KUKA KRL program: MyProgram_118().src

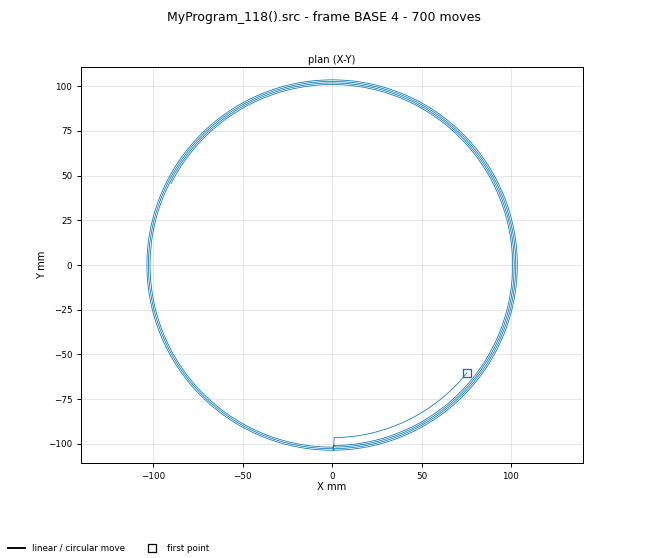
[picture p0: tool path of MyProgram_118().src in frame BASE 4, 700 of 700 moves have a stored position in this frame; points joined in program order, loops and branches not executed]
&ACCESS RVP
&REL 1
&PARAM TEMPLATE = C:\KRC\Roboter\Template\vorgabe
&PARAM EDITMASK = *
DEF MyProgram_118()
; ---- Setting reference (Base) ----
$BASE = BASE_DATA[4]

; --------------------------
; ---- Setting tool (TCP) ----
$TOOL = TOOL_DATA[3]
; --------------------------

$VEL.CP = VEL_APROX_PRINT
Startdeposition()
$VEL.CP = VEL_PRINT
LIN {X 75.3518,Y -60.3472,Z 100,A -43.6794,B 24.9348,C -1.8648,E1 25.1239,E2 129.0277} C_DIS
LIN {X 73.0979,Y -63.0587,Z 100,A -45.771,B 24.9352,C -1.8594,E1 25.1201,E2 131.1226} C_DIS
LIN {X 70.7314,Y -65.7022,Z 100,A -47.8657,B 24.9355,C -1.8545,E1 25.1162,E2 133.2195} C_DIS
LIN {X 68.2631,Y -68.2632,Z 100,A -49.9676,B 24.9359,C -1.8497,E1 25.112,E2 135.324} C_DIS
LIN {X 65.7022,Y -70.7314,Z 100,A -52.0653,B 24.9362,C -1.8452,E1 25.1078,E2 137.4237} C_DIS
LIN {X 63.0587,Y -73.0979,Z 100,A -54.1607,B 24.9365,C -1.8407,E1 25.1034,E2 139.5213} C_DIS
LIN {X 60.3276,Y -75.3677,Z 100,A -56.261,B 24.9368,C -1.8363,E1 25.0988,E2 141.624} C_DIS
LIN {X 57.4574,Y -77.5776,Z 100,A -58.2615,B 24.9368,C -1.8374,E1 25.0944,E2 143.6147} C_DIS
LIN {X 55.5177,Y -78.9773,Z 100,A -59.6429,B 24.9368,C -1.8359,E1 25.0912,E2 144.9948} C_DIS
LIN {X 53.4971,Y -80.3592,Z 100,A -60.9726,B 24.9367,C -1.8377,E1 25.0882,E2 146.3159} C_DIS
LIN {X 51.6359,Y -81.5686,Z 100,A -62.4082,B 24.9372,C -1.8307,E1 25.0848,E2 147.7634} C_DIS
LIN {X 49.5043,Y -82.8788,Z 100,A -63.8332,B 24.9372,C -1.8302,E1 25.0814,E2 149.1851} C_DIS
LIN {X 47.4621,Y -84.065,Z 100,A -65.1647,B 24.9372,C -1.8302,E1 25.0782,E2 150.5124} C_DIS
LIN {X 45.4974,Y -85.1451,Z 100,A -66.5551,B 24.9375,C -1.8257,E1 25.0747,E2 151.9096} C_DIS
LIN {X 43.3997,Y -86.2332,Z 100,A -68.054,B 24.9379,C -1.8198,E1 25.071,E2 153.4184} C_DIS
LIN {X 41.1665,Y -87.3207,Z 100,A -69.422,B 24.9379,C -1.8214,E1 25.0676,E2 154.779} C_DIS
LIN {X 39.1272,Y -88.254,Z 100,A -70.8055,B 24.9381,C -1.8174,E1 25.064,E2 156.1686} C_DIS
LIN {X 36.9553,Y -89.1852,Z 100,A -72.1481,B 24.9381,C -1.8175,E1 25.0606,E2 157.5077} C_DIS
LIN {X 34.7401,Y -90.0713,Z 100,A -73.5591,B 24.9382,C -1.8157,E1 25.0569,E2 158.9197} C_DIS
LIN {X 32.4018,Y -90.9379,Z 100,A -75.1641,B 24.9386,C -1.8092,E1 25.0527,E2 160.5369} C_DIS
LIN {X 29.0265,Y -92.0708,Z 100,A -77.0763,B 24.9383,C -1.814,E1 25.0476,E2 162.4341} C_DIS
LIN {X 26.764,Y -92.7538,Z 100,A -78.5062,B 24.9385,C -1.8114,E1 25.0438,E2 163.8676} C_DIS
LIN {X 24.602,Y -93.3513,Z 100,A -79.929,B 24.9388,C -1.8066,E1 25.0399,E2 165.2995} C_DIS
LIN {X 21.1416,Y -94.1952,Z 100,A -81.9783,B 24.9388,C -1.8069,E1 25.0344,E2 167.3452} C_DIS
LIN {X 18.6908,Y -94.7112,Z 100,A -83.4615,B 24.9388,C -1.8058,E1 25.0303,E2 168.8293} C_DIS
LIN {X 16.3695,Y -95.14,Z 100,A -84.7951,B 24.9388,C -1.8071,E1 25.0267,E2 170.1583} C_DIS
LIN {X 14.0375,Y -95.5119,Z 100,A -86.2601,B 24.939,C -1.8038,E1 25.0226,E2 171.6297} C_DIS
LIN {X 11.6968,Y -95.8268,Z 100,A -87.6386,B 24.939,C -1.8038,E1 25.0188,E2 173.0073} C_DIS
LIN {X 9.2818,Y -96.0905,Z 100,A -89.096,B 24.9391,C -1.8024,E1 25.0147,E2 174.467} C_DIS
LIN {X 7.0631,Y -96.2797,Z 100,A -90.4755,B 24.9393,C -1.7996,E1 25.0109,E2 175.8523} C_DIS
LIN {X 4.7155,Y -96.4233,Z 100,A -92.0156,B 24.9397,C -1.7939,E1 25.0066,E2 177.4054} C_DIS
LIN {X 1.1856,Y -96.5314,Z 100,A -93.9641,B 24.9394,C -1.7985,E1 25.0011,E2 179.3426} C_DIS
LIN {X 1.1856,Y -96.5314,Z 100,A -93.9641,B 24.9394,C -1.7985,E1 25.0011,E2 179.3426} C_DIS
Enddeposition()
LIN {X 0.7197,Y -103.5763,Z 101,A -93.6826,B 24.9456,C -1.7037,E1 25.0013,E2 179.286} C_DIS
Startdeposition()
$VEL.CP = VEL_PRINT
LIN {X -2.1312,Y -103.5571,Z 101,A -95.5889,B 24.9464,C -1.6905,E1 24.9959,E2 181.2235} C_DIS
LIN {X -4.672,Y -103.4736,Z 101,A -96.9948,B 24.9464,C -1.6905,E1 24.992,E2 182.63} C_DIS
LIN {X -7.5389,Y -103.3056,Z 101,A -98.518,B 24.9463,C -1.6929,E1 24.9877,E2 184.1478} C_DIS
LIN {X -9.7436,Y -103.1197,Z 101,A -99.8074,B 24.9464,C -1.6904,E1 24.9841,E2 185.4437} C_DIS
LIN {X -12.6794,Y -102.8018,Z 101,A -101.3905,B 24.9464,C -1.6926,E1 24.9798,E2 187.0228} C_DIS
LIN {X -16.0486,Y -102.3282,Z 101,A -103.2735,B 24.9463,C -1.693,E1 24.9745,E2 188.9063} C_DIS
LIN {X -18.9594,Y -101.8308,Z 101,A -104.9081,B 24.9463,C -1.6935,E1 24.9701,E2 190.5414} C_DIS
LIN {X -21.4527,Y -101.3348,Z 101,A -106.316,B 24.9463,C -1.694,E1 24.9662,E2 191.9497} C_DIS
LIN {X -23.9332,Y -100.7778,Z 101,A -107.7237,B 24.9462,C -1.6947,E1 24.9624,E2 193.3577} C_DIS
LIN {X -26.3992,Y -100.1601,Z 101,A -109.1316,B 24.9462,C -1.6954,E1 24.9586,E2 194.7658} C_DIS
LIN {X -29.674,Y -99.2374,Z 101,A -111.0674,B 24.9462,C -1.6947,E1 24.9534,E2 196.7065} C_DIS
LIN {X -32.9926,Y -98.1838,Z 101,A -113.0237,B 24.9462,C -1.695,E1 24.9481,E2 198.6655} C_DIS
LIN {X -35.7035,Y -97.2311,Z 101,A -114.5894,B 24.946,C -1.6973,E1 24.944,E2 200.2289} C_DIS
LIN {X -38.2402,Y -96.2622,Z 101,A -116.0245,B 24.9458,C -1.7013,E1 24.9403,E2 201.6577} C_DIS
LIN {X -40.81,Y -95.2025,Z 101,A -117.5847,B 24.9458,C -1.702,E1 24.9363,E2 203.2198} C_DIS
LIN {X -44.2865,Y -93.6359,Z 101,A -119.6994,B 24.9456,C -1.7042,E1 24.9309,E2 205.3345} C_DIS
LIN {X -47.3371,Y -92.1293,Z 101,A -121.6373,B 24.9456,C -1.7045,E1 24.9261,E2 207.2769} C_DIS
LIN {X -50.3037,Y -90.5437,Z 101,A -123.5499,B 24.9456,C -1.705,E1 24.9214,E2 209.1935} C_DIS
LIN {X -53.2511,Y -88.8442,Z 101,A -125.4986,B 24.9456,C -1.7053,E1 24.9167,E2 211.1475} C_DIS
LIN {X -56.0379,Y -87.111,Z 101,A -127.1856,B 24.945,C -1.7128,E1 24.9127,E2 212.822} C_DIS
LIN {X -58.2587,Y -85.6419,Z 101,A -128.6912,B 24.945,C -1.714,E1 24.9092,E2 214.3299} C_DIS
LIN {X -60.6774,Y -83.9478,Z 101,A -130.2798,B 24.9447,C -1.7183,E1 24.9056,E2 215.9136} C_DIS
LIN {X -63.4007,Y -81.9083,Z 101,A -132.1691,B 24.9445,C -1.7214,E1 24.9014,E2 217.8023} C_DIS
LIN {X -65.7109,Y -80.069,Z 101,A -133.8091,B 24.9443,C -1.7242,E1 24.8979,E2 219.4419} C_DIS
LIN {X -68.3041,Y -77.8664,Z 101,A -135.6993,B 24.9441,C -1.7275,E1 24.8938,E2 221.3315} C_DIS
LIN {X -70.4972,Y -75.8889,Z 101,A -137.3399,B 24.9439,C -1.7305,E1 24.8905,E2 222.9716} C_DIS
LIN {X -72.3383,Y -74.1359,Z 101,A -138.9245,B 24.9441,C -1.727,E1 24.8873,E2 224.5712} C_DIS
LIN {X -74.6794,Y -71.7745,Z 101,A -140.6694,B 24.9436,C -1.7344,E1 24.8839,E2 226.306} C_DIS
LIN {X -76.4705,Y -69.8633,Z 101,A -142.1075,B 24.9434,C -1.738,E1 24.8811,E2 227.7418} C_DIS
LIN {X -78.4323,Y -67.6561,Z 101,A -143.6981,B 24.943,C -1.7432,E1 24.8782,E2 229.3271} C_DIS
LIN {X -80.055,Y -65.7278,Z 101,A -145.0941,B 24.9428,C -1.7464,E1 24.8757,E2 230.722} C_DIS
LIN {X -81.6575,Y -63.7261,Z 101,A -146.525,B 24.9426,C -1.7493,E1 24.8733,E2 232.1526} C_DIS
LIN {X -83.705,Y -61.0089,Z 101,A -148.3766,B 24.9423,C -1.7551,E1 24.8702,E2 233.9995} C_DIS
LIN {X -85.1771,Y -58.9363,Z 101,A -149.8824,B 24.9423,C -1.7551,E1 24.8678,E2 235.5127} C_DIS
LIN {X -86.8239,Y -56.4852,Z 101,A -151.4738,B 24.9419,C -1.7607,E1 24.8653,E2 237.0986} C_DIS
LIN {X -88.6308,Y -53.6022,Z 101,A -153.3902,B 24.9417,C -1.7644,E1 24.8625,E2 239.0159} C_DIS
LIN {X -90.1243,Y -51.0548,Z 101,A -155.0097,B 24.9413,C -1.7693,E1 24.8602,E2 240.6323} C_DIS
LIN {X -91.3501,Y -48.8276,Z 101,A -156.4246,B 24.9411,C -1.7728,E1 24.8583,E2 242.0462} C_DIS
LIN {X -92.5208,Y -46.5711,Z 101,A -158.0405,B 24.9413,C -1.7693,E1 24.8563,E2 243.6791} C_DIS
LIN {X -93.9989,Y -43.5066,Z 101,A -159.7842,B 24.9406,C -1.7795,E1 24.8542,E2 245.408} C_DIS
LIN {X -95.2025,Y -40.81,Z 101,A -161.3769,B 24.9402,C -1.7856,E1 24.8524,E2 246.9949} C_DIS
LIN {X -96.1753,Y -38.4613,Z 101,A -162.7921,B 24.94,C -1.7894,E1 24.8509,E2 248.4091} C_DIS
LIN {X -97.4033,Y -35.2311,Z 101,A -164.7559,B 24.9397,C -1.7932,E1 24.849,E2 250.3748} C_DIS
LIN {X -98.6509,Y -31.5703,Z 101,A -166.8548,B 24.9392,C -1.801,E1 24.8472,E2 252.4671} C_DIS
LIN {X -99.4821,Y -28.8493,Z 101,A -168.4535,B 24.9389,C -1.8048,E1 24.8459,E2 254.0658} C_DIS
LIN {X -100.1601,Y -26.3992,Z 101,A -169.8694,B 24.9387,C -1.8088,E1 24.8449,E2 255.4805} C_DIS
LIN {X -100.7778,Y -23.9332,Z 101,A -171.2851,B 24.9384,C -1.8128,E1 24.8439,E2 256.895} C_DIS
LIN {X -101.3348,Y -21.4527,Z 101,A -172.7009,B 24.9381,C -1.8168,E1 24.8431,E2 258.3095} C_DIS
LIN {X -101.9831,Y -18.1127,Z 101,A -174.6061,B 24.9378,C -1.8219,E1 24.8421,E2 260.2138} C_DIS
LIN {X -102.4596,Y -15.1985,Z 101,A -176.2405,B 24.9374,C -1.827,E1 24.8414,E2 261.8458} C_DIS
LIN {X -102.8018,Y -12.6794,Z 101,A -177.6567,B 24.9372,C -1.8311,E1 24.8409,E2 263.2606} C_DIS
LIN {X -103.1988,Y -8.8869,Z 101,A -179.7807,B 24.9367,C -1.8373,E1 24.8403,E2 265.3826} C_DIS
LIN {X -103.4333,Y -5.4927,Z 101,A 178.2729,B 24.9365,C -1.8411,E1 24.84,E2 267.3316} C_DIS
LIN {X -103.5369,Y -2.9527,Z 101,A 176.8567,B 24.9362,C -1.8453,E1 24.8398,E2 268.7464} C_DIS
LIN {X -103.5785,Y -0.3823,Z 101,A 175.431,B 24.9359,C -1.8498,E1 24.8398,E2 270.1701} C_DIS
LIN {X -103.5571,Y 2.1312,Z 101,A 174.0243,B 24.9356,C -1.8537,E1 24.8398,E2 271.576} C_DIS
LIN {X -103.4085,Y 5.9414,Z 101,A 171.9,B 24.9352,C -1.86,E1 24.8401,E2 273.698} C_DIS
LIN {X -103.1197,Y 9.7436,Z 101,A 169.8271,B 24.9346,C -1.868,E1 24.8406,E2 275.7641} C_DIS
LIN {X -102.8018,Y 12.6794,Z 101,A 168.1819,B 24.9342,C -1.8729,E1 24.8411,E2 277.4076} C_DIS
LIN {X -102.4596,Y 15.1984,Z 101,A 166.7657,B 24.934,C -1.877,E1 24.8417,E2 278.8223} C_DIS
LIN {X -102.0558,Y 17.7084,Z 101,A 165.3498,B 24.9337,C -1.8812,E1 24.8423,E2 280.2366} C_DIS
LIN {X -101.6681,Y 19.8041,Z 101,A 164.1112,B 24.9335,C -1.8829,E1 24.843,E2 281.4785} C_DIS
LIN {X -101.1515,Y 22.2932,Z 101,A 162.6951,B 24.9332,C -1.8871,E1 24.8438,E2 282.893} C_DIS
LIN {X -100.3261,Y 25.7535,Z 101,A 160.7076,B 24.9328,C -1.8927,E1 24.8451,E2 284.8788} C_DIS
LIN {X -99.5941,Y 28.454,Z 101,A 159.2062,B 24.9324,C -1.8992,E1 24.8462,E2 286.3735} C_DIS
LIN {X -98.7441,Y 31.282,Z 101,A 157.5616,B 24.932,C -1.9039,E1 24.8476,E2 288.0163} C_DIS
LIN {X -97.9467,Y 33.6959,Z 101,A 155.9509,B 24.9322,C -1.9011,E1 24.849,E2 289.6427} C_DIS
LIN {X -96.7856,Y 36.894,Z 101,A 154.1997,B 24.9315,C -1.9115,E1 24.8507,E2 291.379} C_DIS
LIN {X -95.6961,Y 39.6386,Z 101,A 152.6062,B 24.931,C -1.9179,E1 24.8524,E2 292.9662} C_DIS
LIN {X -94.3411,Y 42.7595,Z 101,A 150.7117,B 24.9307,C -1.9232,E1 24.8545,E2 294.8585} C_DIS
LIN {X -93.1341,Y 45.3308,Z 101,A 149.1256,B 24.9304,C -1.9274,E1 24.8564,E2 296.4433} C_DIS
LIN {X -91.9424,Y 47.7029,Z 101,A 147.6523,B 24.9301,C -1.9315,E1 24.8583,E2 297.9145} C_DIS
LIN {X -90.5437,Y 50.3037,Z 101,A 145.9418,B 24.9299,C -1.9336,E1 24.8606,E2 299.629} C_DIS
LIN {X -89.0532,Y 52.8974,Z 101,A 144.3098,B 24.9295,C -1.9392,E1 24.8629,E2 301.2562} C_DIS
LIN {X -87.7282,Y 55.067,Z 101,A 142.8767,B 24.9293,C -1.9423,E1 24.865,E2 302.6893} C_DIS
LIN {X -85.8939,Y 57.8866,Z 101,A 140.9607,B 24.929,C -1.9455,E1 24.8679,E2 304.6071} C_DIS
LIN {X -84.1864,Y 60.3429,Z 101,A 139.3909,B 24.9285,C -1.9531,E1 24.8704,E2 306.1667} C_DIS
LIN {X -82.6801,Y 62.3908,Z 101,A 137.9762,B 24.9282,C -1.9566,E1 24.8728,E2 307.5798} C_DIS
LIN {X -80.8693,Y 64.7234,Z 101,A 136.3333,B 24.9279,C -1.9605,E1 24.8756,E2 309.221} C_DIS
LIN {X -78.6987,Y 67.3434,Z 101,A 134.3892,B 24.9277,C -1.9633,E1 24.8791,E2 311.1676} C_DIS
LIN {X -76.3922,Y 69.9486,Z 101,A 132.4259,B 24.9275,C -1.9668,E1 24.8828,E2 313.1312} C_DIS
LIN {X -74.2252,Y 72.2457,Z 101,A 130.7427,B 24.927,C -1.9733,E1 24.886,E2 314.8061} C_DIS
LIN {X -71.7189,Y 74.7329,Z 101,A 128.734,B 24.9268,C -1.976,E1 24.89,E2 316.8168} C_DIS
LIN {X -69.5606,Y 76.7483,Z 101,A 127.1436,B 24.9264,C -1.9813,E1 24.8933,E2 318.401} C_DIS
LIN {X -67.6561,Y 78.4323,Z 101,A 125.73,B 24.9262,C -1.9843,E1 24.8963,E2 319.8132} C_DIS
LIN {X -65.0426,Y 80.6106,Z 101,A 123.7877,B 24.926,C -1.9863,E1 24.9005,E2 321.758} C_DIS
LIN {X -62.7193,Y 82.4334,Z 101,A 122.1979,B 24.9257,C -1.9913,E1 24.9039,E2 323.3418} C_DIS
LIN {X -59.9771,Y 84.4474,Z 101,A 120.3072,B 24.9254,C -1.9949,E1 24.9082,E2 325.2305} C_DIS
LIN {X -57.5464,Y 86.1242,Z 101,A 118.6668,B 24.9252,C -1.9978,E1 24.912,E2 326.8694} C_DIS
LIN {X -55.4154,Y 87.5106,Z 101,A 117.2545,B 24.925,C -2.0003,E1 24.9153,E2 328.2804} C_DIS
LIN {X -53.2511,Y 88.8442,Z 101,A 115.8427,B 24.9248,C -2.0027,E1 24.9187,E2 329.6909} C_DIS
LIN {X -50.3037,Y 90.5437,Z 101,A 113.9023,B 24.9248,C -2.0039,E1 24.9234,E2 331.6341} C_DIS
LIN {X -47.7029,Y 91.9424,Z 101,A 112.3138,B 24.9244,C -2.0083,E1 24.9273,E2 333.2166} C_DIS
LIN {X -44.2865,Y 93.6359,Z 101,A 110.1968,B 24.9241,C -2.0113,E1 24.9326,E2 335.3318} C_DIS
LIN {X -41.9752,Y 94.6945,Z 101,A 108.7864,B 24.924,C -2.0133,E1 24.9362,E2 336.741} C_DIS
LIN {X -40.0172,Y 95.5366,Z 101,A 107.5526,B 24.924,C -2.013,E1 24.9394,E2 337.9783} C_DIS
LIN {X -36.4737,Y 96.9448,Z 101,A 105.4881,B 24.9237,C -2.0175,E1 24.9447,E2 340.0366} C_DIS
LIN {X -34.0836,Y 97.8107,Z 101,A 104.0778,B 24.9236,C -2.0191,E1 24.9484,E2 341.4458} C_DIS
LIN {X -31.282,Y 98.7441,Z 101,A 102.4402,B 24.9234,C -2.0209,E1 24.9528,E2 343.0822} C_DIS
LIN {X -27.8996,Y 99.7512,Z 101,A 100.457,B 24.9234,C -2.0219,E1 24.9581,E2 345.0663} C_DIS
LIN {X -25.566,Y 100.3743,Z 101,A 99.0933,B 24.9234,C -2.0222,E1 24.9618,E2 346.4312} C_DIS
LIN {X -22.2932,Y 101.1515,Z 101,A 97.1916,B 24.9234,C -2.0224,E1 24.967,E2 348.335} C_DIS
LIN {X -19.3629,Y 101.7531,Z 101,A 95.6221,B 24.923,C -2.0269,E1 24.9712,E2 349.8955} C_DIS
LIN {X -16.4546,Y 102.2654,Z 101,A 93.9858,B 24.9229,C -2.028,E1 24.9757,E2 351.5308} C_DIS
LIN {X -13.5325,Y 102.6912,Z 101,A 92.2602,B 24.9231,C -2.0256,E1 24.9805,E2 353.2634} C_DIS
LIN {X -10.1527,Y 103.082,Z 101,A 90.4658,B 24.9227,C -2.0299,E1 24.9855,E2 355.0488} C_DIS
LIN {X -7.6199,Y 103.3001,Z 101,A 89.0581,B 24.9227,C -2.0305,E1 24.9894,E2 356.4557} C_DIS
LIN {X -3.8125,Y 103.5106,Z 101,A 86.947,B 24.9227,C -2.0311,E1 24.9953,E2 358.5658} C_DIS
LIN {X -1.2711,Y 103.5729,Z 101,A 85.5399,B 24.9227,C -2.0315,E1 24.9992,E2 359.9722} C_DIS
LIN {X 1.2711,Y 103.5729,Z 101,A 84.1332,B 24.9226,C -2.0317,E1 25.0032,E2 361.3783} C_DIS
LIN {X 3.8125,Y 103.5106,Z 101,A 82.7265,B 24.9226,C -2.0318,E1 25.0071,E2 362.7844} C_DIS
LIN {X 6.3516,Y 103.3858,Z 101,A 81.3204,B 24.9226,C -2.0318,E1 25.011,E2 364.1898} C_DIS
LIN {X 9.7436,Y 103.1197,Z 101,A 79.4388,B 24.9226,C -2.0318,E1 25.0162,E2 366.0707} C_DIS
LIN {X 12.6794,Y 102.8018,Z 101,A 77.8057,B 24.9226,C -2.0314,E1 25.0208,E2 367.7033} C_DIS
LIN {X 15.1985,Y 102.4596,Z 101,A 76.4001,B 24.9226,C -2.0311,E1 25.0246,E2 369.1084} C_DIS
LIN {X 17.7084,Y 102.0558,Z 101,A 74.8375,B 24.9231,C -2.0246,E1 25.029,E2 370.6848} C_DIS
LIN {X 20.871,Y 101.4543,Z 101,A 73.1778,B 24.9228,C -2.0285,E1 25.0335,E2 372.3332} C_DIS
LIN {X 23.9332,Y 100.7778,Z 101,A 71.4829,B 24.9228,C -2.0291,E1 25.0381,E2 374.0244} C_DIS
LIN {X 26.3992,Y 100.1601,Z 101,A 70.0787,B 24.9228,C -2.0283,E1 25.0419,E2 375.4284} C_DIS
LIN {X 29.674,Y 99.2374,Z 101,A 68.1779,B 24.923,C -2.0263,E1 25.047,E2 377.3307} C_DIS
LIN {X 32.4914,Y 98.3528,Z 101,A 66.5689,B 24.923,C -2.0259,E1 25.0513,E2 378.9376} C_DIS
LIN {X 34.8953,Y 97.5258,Z 101,A 65.1651,B 24.9231,C -2.0248,E1 25.055,E2 380.3413} C_DIS
LIN {X 38.3932,Y 96.2021,Z 101,A 63.1139,B 24.9232,C -2.0235,E1 25.0603,E2 382.3912} C_DIS
LIN {X 40.81,Y 95.2025,Z 101,A 61.6572,B 24.9234,C -2.0215,E1 25.0641,E2 383.8491} C_DIS
LIN {X 44.2865,Y 93.6359,Z 101,A 59.5533,B 24.9235,C -2.0193,E1 25.0694,E2 385.9529} C_DIS
LIN {X 46.203,Y 92.7033,Z 101,A 58.3266,B 24.9238,C -2.016,E1 25.0725,E2 387.1842} C_DIS
LIN {X 48.4641,Y 91.5415,Z 101,A 56.9245,B 24.9239,C -2.0143,E1 25.076,E2 388.5864} C_DIS
LIN {X 51.0548,Y 90.1243,Z 101,A 55.3466,B 24.9239,C -2.0142,E1 25.0798,E2 390.1599} C_DIS
LIN {X 53.9863,Y 88.3974,Z 101,A 53.4198,B 24.9243,C -2.0096,E1 25.0844,E2 392.0915} C_DIS
LIN {X 56.4852,Y 86.8239,Z 101,A 51.8425,B 24.9243,C -2.0093,E1 25.0881,E2 393.6645} C_DIS
LIN {X 59.6426,Y 84.686,Z 101,A 49.7408,B 24.9245,C -2.0061,E1 25.093,E2 395.7666} C_DIS
LIN {X 62.7193,Y 82.4334,Z 101,A 47.6396,B 24.9248,C -2.0027,E1 25.0977,E2 397.8684} C_DIS
LIN {X 65.7109,Y 80.069,Z 101,A 45.5388,B 24.9251,C -1.9991,E1 25.1023,E2 399.9697} C_DIS
LIN {X 67.6561,Y 78.4323,Z 101,A 44.1385,B 24.9253,C -1.9966,E1 25.1053,E2 401.3705} C_DIS
LIN {X 69.5606,Y 76.7483,Z 101,A 42.7382,B 24.9254,C -1.9941,E1 25.1082,E2 402.7712} C_DIS
LIN {X 71.4231,Y 75.018,Z 101,A 41.1449,B 24.9262,C -1.9836,E1 25.1115,E2 404.3826} C_DIS
LIN {X 73.8472,Y 72.6306,Z 101,A 39.4646,B 24.9259,C -1.9878,E1 25.1147,E2 406.0461} C_DIS
LIN {X 75.8889,Y 70.4972,Z 101,A 37.839,B 24.9262,C -1.9845,E1 25.1179,E2 407.6724} C_DIS
LIN {X 78.162,Y 67.9656,Z 101,A 35.9155,B 24.9266,C -1.9785,E1 25.1214,E2 409.6013} C_DIS
LIN {X 80.069,Y 65.7109,Z 101,A 34.3411,B 24.9267,C -1.9771,E1 25.1242,E2 411.172} C_DIS
LIN {X 81.6575,Y 63.7261,Z 101,A 32.7856,B 24.9274,C -1.9676,E1 25.127,E2 412.7425} C_DIS
LIN {X 83.6393,Y 61.0987,Z 101,A 31.0545,B 24.9274,C -1.9668,E1 25.1298,E2 414.4672} C_DIS
LIN {X 85.4116,Y 58.5989,Z 101,A 29.4454,B 24.9275,C -1.966,E1 25.1324,E2 416.0704} C_DIS
LIN {X 87.1894,Y 55.9157,Z 101,A 27.5793,B 24.9281,C -1.9579,E1 25.1353,E2 417.9463} C_DIS
LIN {X 89.0532,Y 52.8974,Z 101,A 25.6298,B 24.9285,C -1.9532,E1 25.1381,E2 419.8969} C_DIS
LIN {X 90.5437,Y 50.3037,Z 101,A 24.0281,B 24.9286,C -1.9509,E1 25.1403,E2 421.4957} C_DIS
LIN {X 91.9424,Y 47.7029,Z 101,A 22.4548,B 24.9288,C -1.9488,E1 25.1423,E2 423.0656} C_DIS
LIN {X 93.4579,Y 44.6568,Z 101,A 20.5335,B 24.9293,C -1.942,E1 25.1447,E2 424.9927} C_DIS
LIN {X 94.6945,Y 41.9752,Z 101,A 18.9609,B 24.9295,C -1.9398,E1 25.1465,E2 426.562} C_DIS
LIN {X 95.5764,Y 39.9228,Z 101,A 17.7023,B 24.9298,C -1.9353,E1 25.1479,E2 427.8242} C_DIS
LIN {X 96.8206,Y 36.8014,Z 101,A 15.8029,B 24.9303,C -1.9282,E1 25.1498,E2 429.7299} C_DIS
LIN {X 97.8107,Y 34.0836,Z 101,A 14.3109,B 24.9303,C -1.9279,E1 25.1512,E2 431.2143} C_DIS
LIN {X 98.6177,Y 31.6729,Z 101,A 12.8987,B 24.9306,C -1.9234,E1 25.1524,E2 432.629} C_DIS
LIN {X 99.3652,Y 29.2432,Z 101,A 11.4511,B 24.9311,C -1.9174,E1 25.1536,E2 434.0824} C_DIS
LIN {X 100.1601,Y 26.3992,Z 101,A 9.8788,B 24.9313,C -1.915,E1 25.1548,E2 435.6516} C_DIS
LIN {X 101.0445,Y 22.7788,Z 101,A 7.8283,B 24.9317,C -1.9091,E1 25.1561,E2 437.7041} C_DIS
LIN {X 101.5078,Y 20.6101,Z 101,A 6.5622,B 24.9321,C -1.9036,E1 25.1568,E2 438.9757} C_DIS
LIN {X 102.1977,Y 16.8599,Z 101,A 4.4897,B 24.9324,C -1.8985,E1 25.1578,E2 441.048} C_DIS
LIN {X 102.5806,Y 14.3467,Z 101,A 3.1373,B 24.9326,C -1.8963,E1 25.1584,E2 442.3978} C_DIS
LIN {X 102.9018,Y 11.825,Z 101,A 1.6738,B 24.9331,C -1.8894,E1 25.1589,E2 443.8688} C_DIS
LIN {X 103.1988,Y 8.8869,Z 101,A 0.102,B 24.9333,C -1.8868,E1 25.1593,E2 445.4375} C_DIS
LIN {X 103.3581,Y 6.7616,Z 101,A -1.1192,B 24.9337,C -1.8813,E1 25.1595,E2 446.6645} C_DIS
LIN {X 103.5106,Y 3.8125,Z 101,A -2.691,B 24.9338,C -1.8785,E1 25.1597,E2 448.2333} C_DIS
LIN {X 103.5729,Y 1.2711,Z 101,A -4.0799,B 24.9341,C -1.8747,E1 25.1597,E2 449.623} C_DIS
LIN {X 103.5729,Y -1.2711,Z 101,A -5.4839,B 24.9344,C -1.8703,E1 25.1597,E2 451.0291} C_DIS
LIN {X 103.5111,Y -3.7935,Z 101,A -6.8656,B 24.9347,C -1.8664,E1 25.1597,E2 452.4119} C_DIS
LIN {X 103.3858,Y -6.3516,Z 101,A -8.2767,B 24.935,C -1.862,E1 25.1594,E2 453.8248} C_DIS
LIN {X 103.2315,Y -8.4774,Z 101,A -9.498,B 24.9354,C -1.8565,E1 25.1592,E2 455.052} C_DIS
LIN {X 102.8907,Y -11.9203,Z 101,A -11.4317,B 24.9359,C -1.8494,E1 25.1586,E2 456.9908} C_DIS
LIN {X 102.5151,Y -14.8081,Z 101,A -12.9452,B 24.9359,C -1.8483,E1 25.158,E2 458.4981} C_DIS
LIN {X 102.1235,Y -17.3031,Z 101,A -14.3856,B 24.9364,C -1.842,E1 25.1574,E2 459.9449} C_DIS
LIN {X 101.5078,Y -20.6101,Z 101,A -16.2697,B 24.9369,C -1.835,E1 25.1564,E2 461.8343} C_DIS
LIN {X 100.7778,Y -23.9332,Z 101,A -18.0521,B 24.937,C -1.8331,E1 25.1553,E2 463.6109} C_DIS
LIN {X 99.9358,Y -27.2297,Z 101,A -19.9214,B 24.9374,C -1.8277,E1 25.1539,E2 465.4822} C_DIS
LIN {X 99.2374,Y -29.674,Z 101,A -21.3683,B 24.9378,C -1.8216,E1 25.1528,E2 466.9353} C_DIS
LIN {X 98.4793,Y -32.1005,Z 101,A -22.7649,B 24.9381,C -1.8176,E1 25.1516,E2 468.3334} C_DIS
LIN {X 97.2311,Y -35.7035,Z 101,A -24.8603,B 24.9385,C -1.8116,E1 25.1497,E2 470.4313} C_DIS
LIN {X 96.2333,Y -38.3137,Z 101,A -26.3254,B 24.9385,C -1.8101,E1 25.1482,E2 471.8916} C_DIS
LIN {X 95.2025,Y -40.81,Z 101,A -27.8293,B 24.9389,C -1.8051,E1 25.1466,E2 473.3991} C_DIS
LIN {X 93.6359,Y -44.2865,Z 101,A -29.925,B 24.9393,C -1.7993,E1 25.1441,E2 475.4971} C_DIS
LIN {X 92.1293,Y -47.3371,Z 101,A -31.7946,B 24.9397,C -1.7942,E1 25.1418,E2 477.3687} C_DIS
LIN {X 90.9399,Y -49.5838,Z 101,A -33.2427,B 24.9401,C -1.7883,E1 25.1399,E2 478.8231} C_DIS
LIN {X 89.0532,Y -52.8974,Z 101,A -35.3388,B 24.9404,C -1.7828,E1 25.1369,E2 480.9215} C_DIS
LIN {X 87.0459,Y -56.1394,Z 101,A -37.3509,B 24.9406,C -1.7808,E1 25.1339,E2 482.9281} C_DIS
LIN {X 85.6419,Y -58.2587,Z 101,A -38.8328,B 24.941,C -1.7737,E1 25.1316,E2 484.4195} C_DIS
LIN {X 83.9478,Y -60.6774,Z 101,A -40.4063,B 24.9412,C -1.7716,E1 25.1291,E2 485.9901} C_DIS
LIN {X 82.4334,Y -62.7193,Z 101,A -41.804,B 24.9414,C -1.7681,E1 25.1267,E2 487.3894} C_DIS
LIN {X 80.8693,Y -64.7234,Z 101,A -43.3929,B 24.9422,C -1.7569,E1 25.1239,E2 488.9974} C_DIS
LIN {X 78.6987,Y -67.3434,Z 101,A -45.0735,B 24.9419,C -1.7603,E1 25.121,E2 490.6624} C_DIS
LIN {X 77.0223,Y -69.2545,Z 101,A -46.5226,B 24.9423,C -1.7549,E1 25.1183,E2 492.1177} C_DIS
LIN {X 75.2995,Y -71.1238,Z 101,A -47.9212,B 24.9425,C -1.7517,E1 25.1156,E2 493.5178} C_DIS
LIN {X 72.3383,Y -74.1359,Z 101,A -50.1951,B 24.9427,C -1.7485,E1 25.1111,E2 495.7895} C_DIS
LIN {X 70.4972,Y -75.8889,Z 101,A -51.5941,B 24.9429,C -1.7454,E1 25.1083,E2 497.19} C_DIS
LIN {X 68.6135,Y -77.5961,Z 101,A -52.9931,B 24.9431,C -1.7425,E1 25.1053,E2 498.5905} C_DIS
LIN {X 66.6885,Y -79.2566,Z 101,A -54.3924,B 24.9433,C -1.7395,E1 25.1024,E2 499.9912} C_DIS
LIN {X 65.0426,Y -80.6106,Z 101,A -55.6165,B 24.9436,C -1.7351,E1 25.0997,E2 501.2211} C_DIS
LIN {X 62.7193,Y -82.4334,Z 101,A -57.1917,B 24.9436,C -1.7339,E1 25.0962,E2 502.7932} C_DIS
LIN {X 59.9771,Y -84.4474,Z 101,A -59.0654,B 24.9439,C -1.7304,E1 25.092,E2 504.6687} C_DIS
LIN {X 57.5464,Y -86.1242,Z 101,A -60.6917,B 24.9441,C -1.7274,E1 25.0882,E2 506.2967} C_DIS
LIN {X 55.4154,Y -87.5106,Z 101,A -62.0923,B 24.9442,C -1.7249,E1 25.0849,E2 507.6986} C_DIS
LIN {X 52.1569,Y -89.4909,Z 101,A -64.1931,B 24.9445,C -1.7213,E1 25.0799,E2 509.8013} C_DIS
LIN {X 50.3037,Y -90.5437,Z 101,A -65.418,B 24.9447,C -1.7174,E1 25.0769,E2 511.032} C_DIS
LIN {X 47.7029,Y -91.9424,Z 101,A -66.995,B 24.9447,C -1.7168,E1 25.073,E2 512.6058} C_DIS
LIN {X 45.4322,Y -93.0854,Z 101,A -68.3961,B 24.9449,C -1.7147,E1 25.0695,E2 514.008} C_DIS
LIN {X 42.2403,Y -94.5751,Z 101,A -70.3654,B 24.9451,C -1.7109,E1 25.0645,E2 515.9815} C_DIS
LIN {X 40.0172,Y -95.5366,Z 101,A -71.7243,B 24.9453,C -1.7081,E1 25.061,E2 517.3436} C_DIS
LIN {X 36.4737,Y -96.9448,Z 101,A -73.8273,B 24.9455,C -1.7055,E1 25.0555,E2 519.4484} C_DIS
LIN {X 33.6959,Y -97.9467,Z 101,A -75.4057,B 24.9455,C -1.7055,E1 25.0514,E2 521.0234} C_DIS
LIN {X 31.282,Y -98.7441,Z 101,A -76.808,B 24.9455,C -1.704,E1 25.0477,E2 522.4267} C_DIS
LIN {X 28.8493,Y -99.4821,Z 101,A -78.2108,B 24.9457,C -1.7025,E1 25.0439,E2 523.8306} C_DIS
LIN {X 26.3992,Y -100.1601,Z 101,A -79.614,B 24.9457,C -1.7011,E1 25.0401,E2 525.2349} C_DIS
LIN {X 23.9332,Y -100.7778,Z 101,A -81.1742,B 24.9462,C -1.6936,E1 25.0358,E2 526.8105} C_DIS
LIN {X 20.7911,Y -101.4707,Z 101,A -82.8318,B 24.946,C -1.6969,E1 25.0313,E2 528.4583} C_DIS
LIN {X 18.1127,Y -101.9831,Z 101,A -84.3501,B 24.9461,C -1.6953,E1 25.0272,E2 529.9786} C_DIS
LIN {X 15.1985,Y -102.4596,Z 101,A -85.9302,B 24.9461,C -1.6961,E1 25.0228,E2 531.5551} C_DIS
LIN {X 12.6794,Y -102.8018,Z 101,A -87.3346,B 24.9461,C -1.6953,E1 25.0189,E2 532.9604} C_DIS
LIN {X 8.8869,Y -103.1988,Z 101,A -89.4414,B 24.9462,C -1.6942,E1 25.0131,E2 535.0684} C_DIS
LIN {X 5.4927,Y -103.4333,Z 101,A -91.3723,B 24.9464,C -1.6915,E1 25.0077,E2 537.0049} C_DIS
LIN {X 2.9838,Y -103.536,Z 101,A -92.7673,B 24.9464,C -1.6908,E1 25.0038,E2 538.4012} C_DIS
LIN {X 0.7197,Y -103.5763,Z 101,A -93.6825,B 24.9456,C -1.7036,E1 25.0013,E2 539.286} C_DIS
Enddeposition()
LIN {X 0.7197,Y -103.5763,Z 101,A -93.6825,B 24.9456,C -1.7036,E1 25.0013,E2 539.286} C_DIS
Startdeposition()
$VEL.CP = VEL_PRINT
LIN {X 1.2846,Y -102.7027,Z 101,A -92.9534,B 24.9436,C -1.735,E1 25.0035,E2 538.4828} C_DIS
LIN {X 4.3183,Y -102.6182,Z 101,A -91.2193,B 24.9434,C -1.7372,E1 25.0084,E2 536.7437} C_DIS
LIN {X 7.8756,Y -102.4071,Z 101,A -89.234,B 24.9434,C -1.738,E1 25.0139,E2 534.7575} C_DIS
LIN {X 11.1795,Y -102.0999,Z 101,A -87.5018,B 24.9436,C -1.7343,E1 25.0187,E2 533.0351} C_DIS
LIN {X 13.8065,Y -101.7786,Z 101,A -85.7666,B 24.9429,C -1.7455,E1 25.0236,E2 531.2749} C_DIS
LIN {X 17.8429,Y -101.1478,Z 101,A -83.5454,B 24.9429,C -1.7449,E1 25.0297,E2 529.0572} C_DIS
LIN {X 21.9386,Y -100.3386,Z 101,A -81.3604,B 24.9432,C -1.7413,E1 25.0356,E2 526.8836} C_DIS
LIN {X 25.2716,Y -99.5519,Z 101,A -79.3368,B 24.9428,C -1.7477,E1 25.0412,E2 524.8478} C_DIS
LIN {X 28.7194,Y -98.6134,Z 101,A -77.4248,B 24.9428,C -1.7466,E1 25.0463,E2 522.9415} C_DIS
LIN {X 32.5903,Y -97.4016,Z 101,A -75.2957,B 24.943,C -1.744,E1 25.0519,E2 520.8225} C_DIS
LIN {X 35.0796,Y -96.5327,Z 101,A -73.6738,B 24.9425,C -1.752,E1 25.0562,E2 519.185} C_DIS
LIN {X 38.5846,Y -95.1861,Z 101,A -71.5285,B 24.9421,C -1.757,E1 25.0618,E2 517.0328} C_DIS
LIN {X 42.2742,Y -93.6057,Z 101,A -69.3955,B 24.9422,C -1.7561,E1 25.0672,E2 514.9071} C_DIS
LIN {X 44.499,Y -92.5688,Z 101,A -66.9776,B 24.9392,C -1.8011,E1 25.0736,E2 512.3892} C_DIS
LIN {X 49.6708,Y -89.9008,Z 101,A -64.4825,B 24.9409,C -1.7758,E1 25.0795,E2 509.9609} C_DIS
LIN {X 53.3526,Y -87.7647,Z 101,A -62.44,B 24.9415,C -1.7667,E1 25.0844,E2 507.9463} C_DIS
LIN {X 56.0089,Y -86.0959,Z 101,A -60.6502,B 24.9412,C -1.7717,E1 25.0886,E2 506.1506} C_DIS
LIN {X 60.3448,Y -83.1133,Z 101,A -57.3342,B 24.9397,C -1.7933,E1 25.0962,E2 502.795} C_DIS
LIN {X 63.0108,Y -81.1106,Z 101,A -55.9304,B 24.9407,C -1.7785,E1 25.0992,E2 501.4312} C_DIS
LIN {X 64.7275,Y -79.7464,Z 101,A -54.412,B 24.9397,C -1.7934,E1 25.1026,E2 499.8835} C_DIS
LIN {X 68.4218,Y -76.6003,Z 101,A -51.7979,B 24.9396,C -1.7958,E1 25.1081,E2 497.274} C_DIS
LIN {X 72.6951,Y -72.5592,Z 101,A -48.2906,B 24.9384,C -1.8131,E1 25.1152,E2 493.7406} C_DIS
LIN {X 74.9705,Y -70.2028,Z 101,A -46.7603,B 24.9389,C -1.8053,E1 25.118,E2 492.2352} C_DIS
LIN {X 77.9251,Y -66.9088,Z 101,A -44.22,B 24.9383,C -1.8147,E1 25.1227,E2 489.6842} C_DIS
LIN {X 80.5019,Y -63.7855,Z 101,A -42.1577,B 24.9384,C -1.8125,E1 25.1263,E2 487.6367} C_DIS
LIN {X 82.8712,Y -60.6754,Z 101,A -40.0472,B 24.9382,C -1.8155,E1 25.1298,E2 485.5293} C_DIS
LIN {X 84.994,Y -57.6642,Z 101,A -38.2347,B 24.9385,C -1.8111,E1 25.1327,E2 483.7359} C_DIS
LIN {X 86.4611,Y -55.4402,Z 101,A -36.5854,B 24.9378,C -1.8221,E1 25.1352,E2 482.069} C_DIS
LIN {X 89.6902,Y -50.048,Z 101,A -33.1572,B 24.9373,C -1.8289,E1 25.1401,E2 478.6423} C_DIS
LIN {X 91.2491,Y -47.1481,Z 101,A -31.1606,B 24.9365,C -1.841,E1 25.1427,E2 476.6276} C_DIS
LIN {X 92.7997,Y -44.0184,Z 101,A -29.2332,B 24.9361,C -1.846,E1 25.1451,E2 474.6989} C_DIS
LIN {X 94.2495,Y -40.8195,Z 101,A -27.3975,B 24.9361,C -1.8468,E1 25.1471,E2 472.8713} C_DIS
LIN {X 95.8885,Y -36.8069,Z 101,A -24.9257,B 24.9354,C -1.8565,E1 25.1497,E2 470.3903} C_DIS
LIN {X 96.7634,Y -34.4412,Z 101,A -23.1299,B 24.9339,C -1.8772,E1 25.1514,E2 468.5557} C_DIS
LIN {X 97.79,Y -31.4053,Z 101,A -21.7515,B 24.9348,C -1.8656,E1 25.1526,E2 467.2124} C_DIS
LIN {X 98.8014,Y -28.0609,Z 101,A -19.8458,B 24.9345,C -1.87,E1 25.1541,E2 465.3075} C_DIS
LIN {X 99.6341,Y -24.9507,Z 101,A -17.9795,B 24.9338,C -1.8786,E1 25.1554,E2 463.4315} C_DIS
LIN {X 100.5889,Y -20.7611,Z 101,A -15.6435,B 24.9335,C -1.8837,E1 25.1568,E2 461.097} C_DIS
LIN {X 101.3797,Y -16.4774,Z 101,A -13.1519,B 24.9327,C -1.8941,E1 25.158,E2 458.5955} C_DIS
LIN {X 101.9231,Y -12.6919,Z 101,A -11.0307,B 24.9323,C -1.9005,E1 25.1588,E2 456.4718} C_DIS
LIN {X 102.2374,Y -9.8396,Z 101,A -9.6525,B 24.9326,C -1.8963,E1 25.1591,E2 455.1116} C_DIS
LIN {X 102.4393,Y -7.4564,Z 101,A -8.1389,B 24.9317,C -1.9081,E1 25.1595,E2 453.579} C_DIS
LIN {X 102.6202,Y -4.2718,Z 101,A -6.4683,B 24.9317,C -1.9094,E1 25.1597,E2 451.9155} C_DIS
LIN {X 102.7066,Y -0.7114,Z 101,A -4.5432,B 24.9314,C -1.9132,E1 25.1597,E2 449.9928} C_DIS
LIN {X 102.6882,Y 2.0731,Z 101,A -2.9712,B 24.931,C -1.919,E1 25.1597,E2 448.4165} C_DIS
LIN {X 102.5585,Y 5.5588,Z 101,A -1.0552,B 24.9306,C -1.924,E1 25.1595,E2 446.5001} C_DIS
LIN {X 102.3352,Y 8.7742,Z 101,A 0.8717,B 24.9298,C -1.9351,E1 25.1591,E2 444.5584} C_DIS
LIN {X 102.0076,Y 11.9829,Z 101,A 2.5558,B 24.9298,C -1.936,E1 25.1585,E2 442.882} C_DIS
LIN {X 101.5799,Y 15.1961,Z 101,A 4.6086,B 24.9286,C -1.952,E1 25.1577,E2 440.8037} C_DIS
LIN {X 100.8476,Y 19.4651,Z 101,A 6.7502,B 24.9288,C -1.9481,E1 25.1567,E2 438.6839} C_DIS
LIN {X 100.1987,Y 22.5743,Z 101,A 8.66,B 24.928,C -1.9593,E1 25.1555,E2 436.7586} C_DIS
LIN {X 98.0868,Y 30.4651,Z 101,A 12.7741,B 24.9284,C -1.9548,E1 25.1525,E2 432.679} C_DIS
LIN {X 97.053,Y 33.6159,Z 101,A 14.9538,B 24.9269,C -1.974,E1 25.1505,E2 430.4662} C_DIS
LIN {X 95.8124,Y 37.0063,Z 101,A 16.8724,B 24.9268,C -1.9759,E1 25.1486,E2 428.5538} C_DIS
LIN {X 94.3958,Y 40.4838,Z 101,A 19.1718,B 24.9257,C -1.9905,E1 25.1461,E2 426.2326} C_DIS
LIN {X 92.7275,Y 44.1686,Z 101,A 21.2317,B 24.9258,C -1.9888,E1 25.1437,E2 424.1879} C_DIS
LIN {X 91.3053,Y 47.0382,Z 101,A 23.0524,B 24.9254,C -1.9951,E1 25.1414,E2 422.3618} C_DIS
LIN {X 89.7662,Y 49.9119,Z 101,A 24.9635,B 24.9247,C -2.0039,E1 25.1388,E2 420.44} C_DIS
LIN {X 87.9117,Y 53.1106,Z 101,A 26.8115,B 24.925,C -2.0006,E1 25.1362,E2 418.6093} C_DIS
LIN {X 85.9915,Y 56.1676,Z 101,A 29.6011,B 24.9221,C -2.0379,E1 25.1319,E2 415.7457} C_DIS
LIN {X 83.4155,Y 59.9258,Z 101,A 31.4055,B 24.924,C -2.0138,E1 25.1291,E2 414.0069} C_DIS
LIN {X 80.7793,Y 63.4345,Z 101,A 33.8836,B 24.9234,C -2.021,E1 25.1249,E2 411.5235} C_DIS
LIN {X 78.4146,Y 66.3356,Z 101,A 35.831,B 24.9234,C -2.0202,E1 25.1214,E2 409.5871} C_DIS
LIN {X 75.689,Y 69.4285,Z 101,A 38.0011,B 24.9234,C -2.0202,E1 25.1174,E2 407.4268} C_DIS
LIN {X 72.8437,Y 72.4087,Z 101,A 40.5716,B 24.9223,C -2.0361,E1 25.1123,E2 404.8295} C_DIS
LIN {X 69.9569,Y 75.2029,Z 101,A 42.8042,B 24.9219,C -2.0404,E1 25.1078,E2 402.596} C_DIS
LIN {X 67.3874,Y 77.5121,Z 101,A 44.6138,B 24.922,C -2.0395,E1 25.104,E2 400.7957} C_DIS
LIN {X 61.3795,Y 82.3519,Z 101,A 49.0079,B 24.9211,C -2.051,E1 25.0944,E2 396.3909} C_DIS
LIN {X 59.2274,Y 83.9138,Z 101,A 50.724,B 24.9202,C -2.0628,E1 25.0904,E2 394.6527} C_DIS
LIN {X 55.3493,Y 86.5195,Z 101,A 53.0821,B 24.9207,C -2.057,E1 25.085,E2 392.316} C_DIS
LIN {X 52.361,Y 88.3599,Z 101,A 55.2297,B 24.9198,C -2.0675,E1 25.0798,E2 390.1503} C_DIS
LIN {X 48.6547,Y 90.4543,Z 101,A 57.3814,B 24.9203,C -2.0619,E1 25.0746,E2 388.0182} C_DIS
LIN {X 45.5653,Y 92.0486,Z 101,A 59.2397,B 24.9203,C -2.0612,E1 25.07,E2 386.1666} C_DIS
LIN {X 42.1154,Y 93.6773,Z 101,A 61.3542,B 24.9202,C -2.0631,E1 25.0646,E2 384.0528} C_DIS
LIN {X 38.7776,Y 95.1075,Z 101,A 63.3939,B 24.92,C -2.0658,E1 25.0593,E2 382.0116} C_DIS
LIN {X 35.4317,Y 96.4043,Z 101,A 65.0914,B 24.9207,C -2.0559,E1 25.055,E2 380.3413} C_DIS
LIN {X 29.7592,Y 98.3047,Z 101,A 68.7854,B 24.9195,C -2.0724,E1 25.0451,E2 376.6151} C_DIS
LIN {X 26.3905,Y 99.2615,Z 101,A 70.6922,B 24.9195,C -2.0719,E1 25.04,E2 374.7126} C_DIS
LIN {X 22.9615,Y 100.1096,Z 101,A 72.6973,B 24.9193,C -2.0743,E1 25.0345,E2 372.7046} C_DIS
LIN {X 19.6996,Y 100.8025,Z 101,A 74.4976,B 24.9194,C -2.0728,E1 25.0296,E2 370.9101} C_DIS
LIN {X 15.2767,Y 101.5674,Z 101,A 76.9976,B 24.9194,C -2.0735,E1 25.0227,E2 368.411} C_DIS
LIN {X 12.6479,Y 101.9288,Z 101,A 78.5445,B 24.9192,C -2.0764,E1 25.0184,E2 366.8585} C_DIS
LIN {X 9.151,Y 102.3009,Z 101,A 80.4482,B 24.9193,C -2.0744,E1 25.0131,E2 364.9607} C_DIS
LIN {X 5.6258,Y 102.5548,Z 101,A 82.3738,B 24.9194,C -2.0727,E1 25.0078,E2 363.04} C_DIS
LIN {X 2.2805,Y 102.6844,Z 101,A 84.2251,B 24.9195,C -2.0719,E1 25.0026,E2 361.191} C_DIS
LIN {X -1.1823,Y 102.7037,Z 101,A 86.2628,B 24.9192,C -2.0755,E1 24.9969,E2 359.1449} C_DIS
LIN {X -4.6091,Y 102.6057,Z 101,A 88.0371,B 24.9197,C -2.0697,E1 24.992,E2 357.384} C_DIS
LIN {X -7.1397,Y 102.4607,Z 101,A 89.6848,B 24.919,C -2.0779,E1 24.9874,E2 355.7161} C_DIS
LIN {X -10.8726,Y 102.132,Z 101,A 91.6103,B 24.9196,C -2.0706,E1 24.982,E2 353.8069} C_DIS
LIN {X -14.5417,Y 101.6744,Z 101,A 93.6224,B 24.9198,C -2.0675,E1 24.9765,E2 351.8007} C_DIS
LIN {X -18.4713,Y 101.0348,Z 101,A 95.923,B 24.9198,C -2.0688,E1 24.9701,E2 349.4948} C_DIS
LIN {X -21.3687,Y 100.4629,Z 101,A 98.4053,B 24.9174,C -2.0986,E1 24.9632,E2 346.9385} C_DIS
LIN {X -26.1569,Y 99.3243,Z 101,A 100.4019,B 24.9198,C -2.0679,E1 24.958,E2 345.0121} C_DIS
LIN {X -32.0137,Y 97.5932,Z 101,A 103.6549,B 24.9205,C -2.0584,E1 24.9493,E2 341.7762} C_DIS
LIN {X -35.0738,Y 96.5349,Z 101,A 105.5144,B 24.9205,C -2.0581,E1 24.9444,E2 339.9138} C_DIS
LIN {X -37.3986,Y 95.6583,Z 101,A 107.5816,B 24.9188,C -2.0813,E1 24.9389,E2 337.7868} C_DIS
LIN {X -41.2369,Y 94.0675,Z 101,A 108.9061,B 24.9219,C -2.0415,E1 24.9357,E2 336.554} C_DIS
LIN {X -45.8329,Y 91.9159,Z 101,A 111.558,B 24.9227,C -2.0306,E1 24.9291,E2 333.9214} C_DIS
LIN {X -49.2511,Y 90.1308,Z 101,A 114.3045,B 24.9213,C -2.0484,E1 24.9222,E2 331.1248} C_DIS
LIN {X -51.9995,Y 88.5736,Z 101,A 116.0524,B 24.9216,C -2.0448,E1 24.9179,E2 329.3803} C_DIS
LIN {X -54.833,Y 86.8489,Z 101,A 117.7962,B 24.9222,C -2.0375,E1 24.9138,E2 327.6484} C_DIS
LIN {X -56.4788,Y 85.7863,Z 101,A 119.894,B 24.9195,C -2.0719,E1 24.9088,E2 325.4618} C_DIS
LIN {X -60.7228,Y 82.8364,Z 101,A 122.0691,B 24.9219,C -2.0402,E1 24.904,E2 323.3545} C_DIS
LIN {X -63.4589,Y 80.7601,Z 101,A 123.7632,B 24.9229,C -2.0281,E1 24.9003,E2 321.683} C_DIS
LIN {X -65.3935,Y 79.2019,Z 101,A 125.436,B 24.9223,C -2.0354,E1 24.8966,E2 319.9866} C_DIS
LIN {X -68.7473,Y 76.3089,Z 101,A 127.7876,B 24.9231,C -2.0255,E1 24.8917,E2 317.6492} C_DIS
LIN {X -70.7213,Y 74.484,Z 101,A 129.3456,B 24.9231,C -2.024,E1 24.8886,E2 316.0884} C_DIS
LIN {X -73.6059,Y 71.6348,Z 101,A 131.2999,B 24.9244,C -2.0076,E1 24.8848,E2 314.1649} C_DIS
LIN {X -76.1439,Y 68.9316,Z 101,A 133.5821,B 24.9242,C -2.01,E1 24.8804,E2 311.867} C_DIS
LIN {X -78.0995,Y 66.7054,Z 101,A 135.2292,B 24.9246,C -2.0056,E1 24.8774,E2 310.2229} C_DIS
LIN {X -80.3774,Y 63.9431,Z 101,A 137.1655,B 24.9251,C -1.9981,E1 24.874,E2 308.2953} C_DIS
LIN {X -83.9569,Y 59.1647,Z 101,A 140.3786,B 24.9261,C -1.9849,E1 24.8687,E2 305.0981} C_DIS
LIN {X -85.5921,Y 56.7732,Z 101,A 142.077,B 24.9262,C -1.9833,E1 24.8661,E2 303.3951} C_DIS
LIN {X -87.0644,Y 54.4878,Z 101,A 143.7292,B 24.9262,C -1.9838,E1 24.8636,E2 301.7334} C_DIS
LIN {X -88.9006,Y 51.4385,Z 101,A 145.5978,B 24.9269,C -1.974,E1 24.8609,E2 299.8785} C_DIS
LIN {X -90.2513,Y 49.029,Z 101,A 147.2708,B 24.9269,C -1.9742,E1 24.8587,E2 298.1964} C_DIS
LIN {X -91.4733,Y 46.7095,Z 101,A 149.0527,B 24.9264,C -1.9811,E1 24.8564,E2 296.3884} C_DIS
LIN {X -93.6434,Y 42.1907,Z 101,A 151.5519,B 24.9278,C -1.9622,E1 24.8534,E2 293.9206} C_DIS
LIN {X -94.8995,Y 39.288,Z 101,A 153.4043,B 24.928,C -1.9599,E1 24.8514,E2 292.0635} C_DIS
LIN {X -96.0422,Y 36.4011,Z 101,A 155.0694,B 24.9285,C -1.9522,E1 24.8498,E2 290.4072} C_DIS
LIN {X -97.3191,Y 32.8347,Z 101,A 157.1994,B 24.929,C -1.9463,E1 24.8478,E2 288.2794} C_DIS
LIN {X -98.3771,Y 29.5157,Z 101,A 158.9752,B 24.9299,C -1.9343,E1 24.8464,E2 286.5219} C_DIS
LIN {X -99.0066,Y 27.334,Z 101,A 160.6047,B 24.9292,C -1.943,E1 24.8451,E2 284.8623} C_DIS
LIN {X -99.7629,Y 24.4233,Z 101,A 162.0892,B 24.9301,C -1.9309,E1 24.8441,E2 283.3979} C_DIS
LIN {X -100.4701,Y 21.3356,Z 101,A 163.819,B 24.9306,C -1.924,E1 24.8431,E2 281.6745} C_DIS
LIN {X -101.6153,Y 14.9572,Z 101,A 167.6058,B 24.931,C -1.9183,E1 24.8413,E2 277.8788} C_DIS
LIN {X -102.1045,Y 11.1351,Z 101,A 169.539,B 24.9321,C -1.9038,E1 24.8406,E2 275.9685} C_DIS
LIN {X -102.3732,Y 8.2995,Z 101,A 171.3062,B 24.932,C -1.9049,E1 24.8402,E2 274.1881} C_DIS
LIN {X -102.5953,Y 4.8508,Z 101,A 173.3083,B 24.9322,C -1.9013,E1 24.8399,E2 272.1826} C_DIS
LIN {X -102.6969,Y 1.599,Z 101,A 175.1776,B 24.9325,C -1.8974,E1 24.8398,E2 270.3114} C_DIS
LIN {X -102.6811,Y -2.4619,Z 101,A 177.4549,B 24.933,C -1.8905,E1 24.8398,E2 268.0369} C_DIS
LIN {X -102.5322,Y -6.0339,Z 101,A 179.2893,B 24.9339,C -1.8785,E1 24.8401,E2 266.22} C_DIS
LIN {X -102.3231,Y -8.9105,Z 101,A -178.5707,B 24.9329,C -1.892,E1 24.8407,E2 264.0349} C_DIS
LIN {X -101.986,Y -12.1668,Z 101,A -177.2422,B 24.9345,C -1.8687,E1 24.8411,E2 262.754} C_DIS
LIN {X -101.5459,Y -15.4158,Z 101,A -175.6064,B 24.9354,C -1.8562,E1 24.8417,E2 261.1384} C_DIS
LIN {X -100.9486,Y -18.9405,Z 101,A -173.2338,B 24.9349,C -1.8631,E1 24.8429,E2 258.735} C_DIS
LIN {X -100.171,Y -22.6957,Z 101,A -171.1267,B 24.9355,C -1.8554,E1 24.8441,E2 256.6341} C_DIS
LIN {X -99.3437,Y -26.0815,Z 101,A -169.0938,B 24.9357,C -1.8525,E1 24.8455,E2 254.5961} C_DIS
LIN {X -98.3925,Y -29.4639,Z 101,A -167.2372,B 24.9363,C -1.843,E1 24.8469,E2 252.7516} C_DIS
LIN {X -97.3708,Y -32.6816,Z 101,A -165.303,B 24.9366,C -1.8391,E1 24.8486,E2 250.8155} C_DIS
LIN {X -96.2093,Y -35.9597,Z 101,A -163.581,B 24.9375,C -1.8257,E1 24.8502,E2 249.1158} C_DIS
LIN {X -95.2699,Y -38.3786,Z 101,A -161.1502,B 24.9354,C -1.8564,E1 24.8529,E2 246.598} C_DIS
LIN {X -93.4191,Y -42.6874,Z 101,A -159.1131,B 24.9373,C -1.8283,E1 24.8551,E2 244.6169} C_DIS
LIN {X -91.6266,Y -46.4095,Z 101,A -156.9819,B 24.9382,C -1.8157,E1 24.8578,E2 242.5043} C_DIS
LIN {X -90.0978,Y -49.3121,Z 101,A -155.1712,B 24.9386,C -1.81,E1 24.8601,E2 240.6976} C_DIS
LIN {X -88.4473,Y -52.2132,Z 101,A -153.2846,B 24.9389,C -1.8059,E1 24.8628,E2 238.811} C_DIS
LIN {X -86.795,Y -54.9192,Z 101,A -151.3851,B 24.9389,C -1.8059,E1 24.8656,E2 236.9017} C_DIS
LIN {X -85.1039,Y -57.502,Z 101,A -149.712,B 24.9393,C -1.7998,E1 24.8682,E2 235.2349} C_DIS
LIN {X -82.9892,Y -60.5141,Z 101,A -147.6961,B 24.9397,C -1.7933,E1 24.8715,E2 233.2245} C_DIS
LIN {X -80.9618,Y -63.2032,Z 101,A -145.7365,B 24.9398,C -1.7916,E1 24.8748,E2 231.2596} C_DIS
LIN {X -78.7773,Y -65.9043,Z 101,A -143.833,B 24.9402,C -1.7859,E1 24.8782,E2 229.361} C_DIS
LIN {X -76.7165,Y -68.292,Z 101,A -142.2975,B 24.941,C -1.7738,E1 24.881,E2 227.8474} C_DIS
LIN {X -75.137,Y -70.027,Z 101,A -140.7489,B 24.9406,C -1.7795,E1 24.8839,E2 226.2782} C_DIS
LIN {X -72.984,Y -72.2667,Z 101,A -139.0332,B 24.9409,C -1.7752,E1 24.8873,E2 224.5655} C_DIS
LIN {X -70.1547,Y -75.0169,Z 101,A -136.7971,B 24.9412,C -1.7719,E1 24.8918,E2 222.3279} C_DIS
LIN {X -68.0467,Y -76.9361,Z 101,A -134.782,B 24.9403,C -1.7843,E1 24.8961,E2 220.2753} C_DIS
LIN {X -65.5895,Y -79.039,Z 101,A -132.9889,B 24.9406,C -1.7806,E1 24.8999,E2 218.4844} C_DIS
LIN {X -62.9991,Y -81.1196,Z 101,A -131.5641,B 24.9419,C -1.7614,E1 24.903,E2 217.0999} C_DIS
LIN {X -60.621,Y -82.911,Z 101,A -129.9038,B 24.942,C -1.7585,E1 24.9067,E2 215.4406} C_DIS
LIN {X -57.8692,Y -84.8552,Z 101,A -127.9542,B 24.942,C -1.758,E1 24.9112,E2 213.4856} C_DIS
LIN {X -54.8054,Y -86.8661,Z 101,A -125.4894,B 24.9413,C -1.7704,E1 24.9171,E2 210.9834} C_DIS
LIN {X -51.8996,Y -88.6327,Z 101,A -123.9999,B 24.9424,C -1.7525,E1 24.9206,E2 209.532} C_DIS
LIN {X -48.7769,Y -90.388,Z 101,A -121.9672,B 24.9425,C -1.7511,E1 24.9255,E2 207.4967} C_DIS
LIN {X -45.1346,Y -92.2621,Z 101,A -119.7945,B 24.943,C -1.744,E1 24.9309,E2 205.3351} C_DIS
LIN {X -41.859,Y -93.7928,Z 101,A -117.6772,B 24.9429,C -1.7455,E1 24.9363,E2 203.2091} C_DIS
LIN {X -38.8924,Y -95.0608,Z 101,A -115.9608,B 24.9432,C -1.7405,E1 24.9407,E2 201.5006} C_DIS
LIN {X -32.7269,Y -97.3555,Z 101,A -112.3224,B 24.9435,C -1.736,E1 24.9503,E2 197.8655} C_DIS
LIN {X -29.8202,Y -98.2864,Z 101,A -110.4837,B 24.9433,C -1.7399,E1 24.9552,E2 196.0144} C_DIS
LIN {X -26.7483,Y -99.1648,Z 101,A -108.7474,B 24.9435,C -1.737,E1 24.9599,E2 194.2822} C_DIS
LIN {X -23.2674,Y -100.0389,Z 101,A -106.732,B 24.9435,C -1.7365,E1 24.9653,E2 192.2654} C_DIS
LIN {X -20.12,Y -100.7205,Z 101,A -104.8542,B 24.9433,C -1.7388,E1 24.9705,E2 190.3799} C_DIS
LIN {X -16.961,Y -101.2989,Z 101,A -103.1865,B 24.9437,C -1.7335,E1 24.9751,E2 188.7231} C_DIS
LIN {X -13.5988,Y -101.8055,Z 101,A -101.1327,B 24.9433,C -1.7391,E1 24.9808,E2 186.6544} C_DIS
LIN {X -9.6725,Y -102.2528,Z 101,A -99.0035,B 24.9435,C -1.736,E1 24.9867,E2 184.5313} C_DIS
LIN {X -6.3425,Y -102.5146,Z 101,A -97.0749,B 24.9434,C -1.7385,E1 24.9921,E2 182.5961} C_DIS
LIN {X -3.0041,Y -102.6651,Z 101,A -95.3939,B 24.9438,C -1.7316,E1 24.9967,E2 180.9311} C_DIS
LIN {X 0.2157,Y -102.7096,Z 101,A -93.7223,B 24.9441,C -1.7271,E1 25.0013,E2 179.2701} C_DIS
LIN {X 0.2157,Y -102.7096,Z 101,A -93.7223,B 24.9441,C -1.7271,E1 25.0013,E2 179.2701} C_DIS
Enddeposition()
LIN {X 0.7116,Y -101.8367,Z 101,A -94.1279,B 24.9448,C -1.7162,E1 25.0001,E2 179.7015} C_DIS
Startdeposition()
$VEL.CP = VEL_PRINT
LIN {X -2.1922,Y -101.8161,Z 101,A -95.7892,B 24.9448,C -1.7149,E1 24.9955,E2 181.3661} C_DIS
LIN {X -5.9215,Y -101.6673,Z 101,A -97.8011,B 24.9447,C -1.718,E1 24.9899,E2 183.3711} C_DIS
LIN {X -9.0007,Y -101.4413,Z 101,A -99.6463,B 24.9449,C -1.714,E1 24.9847,E2 185.2266} C_DIS
LIN {X -12.2685,Y -101.0984,Z 101,A -101.5049,B 24.9449,C -1.7139,E1 24.9796,E2 187.0867} C_DIS
LIN {X -16.0991,Y -100.5601,Z 101,A -103.6246,B 24.9448,C -1.7165,E1 24.9737,E2 189.2019} C_DIS
LIN {X -20.8865,Y -99.6752,Z 101,A -106.2507,B 24.9444,C -1.7218,E1 24.9666,E2 191.8183} C_DIS
LIN {X -23.883,Y -98.9994,Z 101,A -108.1401,B 24.9448,C -1.7167,E1 24.9614,E2 193.7224} C_DIS
LIN {X -27.4082,Y -98.0823,Z 101,A -110.6108,B 24.9457,C -1.7024,E1 24.9546,E2 196.2308} C_DIS
LIN {X -30.7645,Y -97.083,Z 101,A -112.0073,B 24.9442,C -1.7249,E1 24.951,E2 197.5761} C_DIS
LIN {X -33.4746,Y -96.1808,Z 101,A -114.3974,B 24.946,C -1.6977,E1 24.9446,E2 200.0358} C_DIS
LIN {X -37.4274,Y -94.7125,Z 101,A -115.5922,B 24.9431,C -1.743,E1 24.9417,E2 201.1253} C_DIS
LIN {X -39.5965,Y -93.8261,Z 101,A -117.372,B 24.9441,C -1.7273,E1 24.937,E2 202.9464} C_DIS
LIN {X -42.0293,Y -92.762,Z 101,A -118.8621,B 24.944,C -1.7291,E1 24.9332,E2 204.4359} C_DIS
LIN {X -44.5986,Y -91.5554,Z 101,A -120.9721,B 24.945,C -1.7124,E1 24.9278,E2 206.5909} C_DIS
LIN {X -47.5439,Y -90.06,Z 101,A -122.9275,B 24.9451,C -1.7114,E1 24.9229,E2 208.5543} C_DIS
LIN {X -50.7954,Y -88.2669,Z 101,A -125.0006,B 24.9449,C -1.7149,E1 24.9179,E2 210.6252} C_DIS
LIN {X -53.9073,Y -86.4015,Z 101,A -126.5411,B 24.9435,C -1.7359,E1 24.9144,E2 212.1204} C_DIS
LIN {X -56.8551,Y -84.4914,Z 101,A -128.5511,B 24.9435,C -1.7378,E1 24.9097,E2 214.1325} C_DIS
LIN {X -59.7388,Y -82.4789,Z 101,A -130.636,B 24.9435,C -1.7373,E1 24.9049,E2 216.2258} C_DIS
LIN {X -63.4027,Y -79.6956,Z 101,A -134.0429,B 24.945,C -1.7131,E1 24.8973,E2 219.7029} C_DIS
LIN {X -67.4799,Y -76.2761,Z 101,A -135.9934,B 24.9422,C -1.7557,E1 24.8934,E2 221.5597} C_DIS
LIN {X -70.862,Y -73.1427,Z 101,A -138.8126,B 24.9424,C -1.753,E1 24.8876,E2 224.3968} C_DIS
LIN {X -73.3931,Y -70.6023,Z 101,A -140.6754,B 24.9418,C -1.7628,E1 24.884,E2 226.2442} C_DIS
LIN {X -76.1499,Y -67.6208,Z 101,A -143.0334,B 24.9416,C -1.7653,E1 24.8795,E2 228.6067} C_DIS
LIN {X -78.2981,Y -65.1201,Z 101,A -144.9179,B 24.9414,C -1.7686,E1 24.8761,E2 230.4921} C_DIS
LIN {X -80.6981,Y -62.1212,Z 101,A -147.1256,B 24.9411,C -1.7721,E1 24.8723,E2 232.7017} C_DIS
LIN {X -82.8683,Y -59.1952,Z 101,A -149.1088,B 24.9406,C -1.7795,E1 24.8691,E2 234.677} C_DIS
LIN {X -85.0296,Y -56.0462,Z 101,A -151.2189,B 24.9402,C -1.7863,E1 24.8658,E2 236.7813} C_DIS
LIN {X -86.6891,Y -53.4469,Z 101,A -153.3299,B 24.9408,C -1.7778,E1 24.8626,E2 238.9235} C_DIS
LIN {X -88.9503,Y -49.589,Z 101,A -155.5288,B 24.9396,C -1.7955,E1 24.8596,E2 241.0915} C_DIS
LIN {X -90.5969,Y -46.513,Z 101,A -157.5688,B 24.9394,C -1.7983,E1 24.857,E2 243.1358} C_DIS
LIN {X -92.1061,Y -43.4506,Z 101,A -159.9966,B 24.9402,C -1.7862,E1 24.854,E2 245.6055} C_DIS
LIN {X -93.6087,Y -40.1123,Z 101,A -161.4423,B 24.9384,C -1.8132,E1 24.8524,E2 246.9949} C_DIS
LIN {X -95.3228,Y -35.8447,Z 101,A -163.6655,B 24.937,C -1.8333,E1 24.8502,E2 249.1825} C_DIS
LIN {X -96.1154,Y -33.661,Z 101,A -165.4209,B 24.9378,C -1.8217,E1 24.8485,E2 250.9757} C_DIS
LIN {X -97.5475,Y -29.2539,Z 101,A -167.9953,B 24.9372,C -1.8306,E1 24.8463,E2 253.5435} C_DIS
LIN {X -98.3323,Y -26.4949,Z 101,A -169.7558,B 24.9372,C -1.8306,E1 24.845,E2 255.3145} C_DIS
LIN {X -99.2246,Y -22.928,Z 101,A -171.795,B 24.9367,C -1.8379,E1 24.8436,E2 257.348} C_DIS
LIN {X -99.9775,Y -19.384,Z 101,A -173.8718,B 24.9363,C -1.8429,E1 24.8425,E2 259.425} C_DIS
LIN {X -100.9028,Y -13.7889,Z 101,A -177.0999,B 24.9357,C -1.8517,E1 24.8411,E2 262.6515} C_DIS
LIN {X -101.519,Y -8.0695,Z 101,A 179.7251,B 24.9349,C -1.8641,E1 24.8402,E2 265.8159} C_DIS
LIN {X -101.7329,Y -4.659,Z 101,A 177.2853,B 24.9357,C -1.8527,E1 24.8399,E2 268.2975} C_DIS
LIN {X -101.8337,Y -1.2098,Z 101,A 175.1382,B 24.9357,C -1.852,E1 24.8398,E2 270.4592} C_DIS
LIN {X -101.8001,Y 2.8368,Z 101,A 173.554,B 24.9336,C -1.8827,E1 24.8398,E2 271.9797} C_DIS
LIN {X -101.6681,Y 5.9071,Z 101,A 171.5029,B 24.9339,C -1.8774,E1 24.8402,E2 274.0558} C_DIS
LIN {X -101.0776,Y 12.4456,Z 101,A 168.1341,B 24.9323,C -1.9003,E1 24.8411,E2 277.3902} C_DIS
LIN {X -100.733,Y 14.9805,Z 101,A 166.4209,B 24.9326,C -1.8956,E1 24.8418,E2 279.1247} C_DIS
LIN {X -99.7561,Y 20.4925,Z 101,A 163.3746,B 24.9317,C -1.9093,E1 24.8434,E2 282.1566} C_DIS
LIN {X -98.8667,Y 24.427,Z 101,A 161.2895,B 24.9307,C -1.9227,E1 24.8447,E2 284.2218} C_DIS
LIN {X -98.0736,Y 27.4389,Z 101,A 159.1493,B 24.9312,C -1.9151,E1 24.8463,E2 286.3927} C_DIS
LIN {X -96.8795,Y 31.3938,Z 101,A 156.9983,B 24.9303,C -1.9283,E1 24.848,E2 288.5246} C_DIS
LIN {X -95.6405,Y 34.9874,Z 101,A 154.7785,B 24.93,C -1.9321,E1 24.8501,E2 290.7477} C_DIS
LIN {X -94.3335,Y 38.3721,Z 101,A 152.7971,B 24.9294,C -1.9404,E1 24.8521,E2 292.7204} C_DIS
LIN {X -92.6354,Y 42.3103,Z 101,A 150.5297,B 24.9285,C -1.9527,E1 24.8547,E2 294.9711} C_DIS
LIN {X -89.8023,Y 48.0318,Z 101,A 146.8934,B 24.9278,C -1.9618,E1 24.8592,E2 298.6051} C_DIS
LIN {X -88.3947,Y 50.573,Z 101,A 145.1229,B 24.9278,C -1.9619,E1 24.8616,E2 300.3847} C_DIS
LIN {X -86.6183,Y 53.5602,Z 101,A 143.0877,B 24.9276,C -1.9648,E1 24.8646,E2 302.4236} C_DIS
LIN {X -83.7964,Y 57.8746,Z 101,A 140.1726,B 24.9271,C -1.9724,E1 24.8691,E2 305.3351} C_DIS
LIN {X -80.562,Y 62.2977,Z 101,A 137.5439,B 24.9253,C -1.9964,E1 24.8734,E2 307.9193} C_DIS
LIN {X -79.0081,Y 64.257,Z 101,A 135.2454,B 24.9273,C -1.9694,E1 24.8775,E2 310.2928} C_DIS
LIN {X -76.7921,Y 66.8896,Z 101,A 132.8656,B 24.928,C -1.9592,E1 24.882,E2 312.7076} C_DIS
LIN {X -73.3442,Y 70.653,Z 101,A 131.2919,B 24.9242,C -2.011,E1 24.8848,E2 314.1649} C_DIS
LIN {X -71.6601,Y 72.3606,Z 101,A 128.9512,B 24.9265,C -1.9799,E1 24.8896,E2 316.5894} C_DIS
LIN {X -68.8824,Y 75.0096,Z 101,A 126.3668,B 24.9272,C -1.9704,E1 24.895,E2 319.2069} C_DIS
LIN {X -64.76,Y 78.5973,Z 101,A 124.3738,B 24.9239,C -2.0145,E1 24.899,E2 321.1025} C_DIS
LIN {X -62.5054,Y 80.402,Z 101,A 122.5503,B 24.9242,C -2.0111,E1 24.9031,E2 322.9409} C_DIS
LIN {X -60.1274,Y 82.1944,Z 101,A 120.9635,B 24.9237,C -2.0177,E1 24.9066,E2 324.5177} C_DIS
LIN {X -55.7542,Y 85.2222,Z 101,A 118.0309,B 24.9231,C -2.0257,E1 24.9133,E2 327.4411} C_DIS
LIN {X -53.0133,Y 86.953,Z 101,A 116.1065,B 24.9231,C -2.0255,E1 24.9179,E2 329.3719} C_DIS
LIN {X -49.6786,Y 88.9003,Z 101,A 113.9243,B 24.9228,C -2.0291,E1 24.9232,E2 331.5521} C_DIS
LIN {X -46.3751,Y 90.6674,Z 101,A 111.8225,B 24.9225,C -2.0328,E1 24.9284,E2 333.6508} C_DIS
LIN {X -42.8064,Y 92.406,Z 101,A 109.6443,B 24.9221,C -2.0382,E1 24.9339,E2 335.8217} C_DIS
LIN {X -39.4805,Y 93.875,Z 101,A 107.2902,B 24.9227,C -2.0303,E1 24.94,E2 338.2002} C_DIS
LIN {X -36.1085,Y 95.2229,Z 101,A 105.488,B 24.9218,C -2.0416,E1 24.9446,E2 339.9794} C_DIS
LIN {X -32.7541,Y 96.4284,Z 101,A 102.9751,B 24.923,C -2.026,E1 24.9513,E2 342.5342} C_DIS
LIN {X -29.3755,Y 97.5114,Z 101,A 101.6616,B 24.921,C -2.0527,E1 24.9547,E2 343.7866} C_DIS
LIN {X -27.2509,Y 98.1269,Z 101,A 99.5754,B 24.9232,C -2.0238,E1 24.9605,E2 345.9448} C_DIS
LIN {X -23.3519,Y 99.1257,Z 101,A 97.8406,B 24.9216,C -2.0449,E1 24.9651,E2 347.6316} C_DIS
LIN {X -20.7872,Y 99.6956,Z 101,A 95.4604,B 24.924,C -2.0137,E1 24.9718,E2 350.0886} C_DIS
LIN {X -15.3844,Y 100.6706,Z 101,A 93.4418,B 24.9208,C -2.0545,E1 24.9771,E2 352.0123} C_DIS
LIN {X -12.1526,Y 101.112,Z 101,A 90.8526,B 24.9229,C -2.0282,E1 24.9844,E2 354.6657} C_DIS
LIN {X -7.9328,Y 101.5299,Z 101,A 88.8594,B 24.9217,C -2.0435,E1 24.9899,E2 356.6234} C_DIS
LIN {X -3.5092,Y 101.7794,Z 101,A 86.6469,B 24.9208,C -2.0547,E1 24.996,E2 358.81} C_DIS
LIN {X -0.3729,Y 101.8388,Z 101,A 84.958,B 24.9206,C -2.0579,E1 25.0007,E2 360.4914} C_DIS
LIN {X 3.3537,Y 101.7842,Z 101,A 82.7399,B 24.9209,C -2.0537,E1 25.0069,E2 362.7191} C_DIS
LIN {X 6.5919,Y 101.626,Z 101,A 80.8897,B 24.9209,C -2.0527,E1 25.0121,E2 364.5708} C_DIS
LIN {X 9.9484,Y 101.3536,Z 101,A 78.7867,B 24.9216,C -2.0448,E1 25.018,E2 366.6915} C_DIS
LIN {X 14.7296,Y 100.7692,Z 101,A 75.8454,B 24.9223,C -2.0355,E1 25.0262,E2 369.6523} C_DIS
LIN {X 18.2689,Y 100.1874,Z 101,A 74.4342,B 24.9206,C -2.0575,E1 25.0299,E2 371.0099} C_DIS
LIN {X 21.3567,Y 99.5753,Z 101,A 72.4574,B 24.9213,C -2.0489,E1 25.0353,E2 373.0045} C_DIS
LIN {X 24.0461,Y 98.9596,Z 101,A 70.4954,B 24.9225,C -2.0326,E1 25.0408,E2 375.0022} C_DIS
LIN {X 27.6023,Y 98.0273,Z 101,A 69.1868,B 24.9204,C -2.0599,E1 25.0441,E2 376.2439} C_DIS
LIN {X 30.481,Y 97.1706,Z 101,A 66.5754,B 24.9232,C -2.0238,E1 25.0513,E2 378.9364} C_DIS
LIN {X 34.5969,Y 95.783,Z 101,A 65.0867,B 24.9206,C -2.0578,E1 25.055,E2 380.3413} C_DIS
LIN {X 38.1851,Y 94.4096,Z 101,A 62.5775,B 24.9218,C -2.0424,E1 25.0616,E2 382.8816} C_DIS
LIN {X 41.7107,Y 92.9056,Z 101,A 60.2029,B 24.9226,C -2.0316,E1 25.0677,E2 385.2759} C_DIS
LIN {X 45.2675,Y 91.2254,Z 101,A 58.354,B 24.9217,C -2.0429,E1 25.0723,E2 387.0932} C_DIS
LIN {X 51.4708,Y 87.8757,Z 101,A 54.5211,B 24.9217,C -2.0426,E1 25.0817,E2 390.9157} C_DIS
LIN {X 54.218,Y 86.2074,Z 101,A 52.4588,B 24.9227,C -2.03,E1 25.0866,E2 393.0013} C_DIS
LIN {X 58.6337,Y 83.2687,Z 101,A 49.6866,B 24.9225,C -2.0333,E1 25.093,E2 395.7564} C_DIS
LIN {X 61.1304,Y 81.4511,Z 101,A 46.8665,B 24.9259,C -1.9882,E1 25.0995,E2 398.6729} C_DIS
LIN {X 65.4372,Y 78.0346,Z 101,A 44.8633,B 24.9231,C -2.0248,E1 25.1036,E2 400.5821} C_DIS
LIN {X 67.8813,Y 75.9168,Z 101,A 42.9965,B 24.9235,C -2.0193,E1 25.1075,E2 402.4543} C_DIS
LIN {X 70.4388,Y 73.5506,Z 101,A 40.9772,B 24.924,C -2.0129,E1 25.1116,E2 404.4804} C_DIS
LIN {X 72.8276,Y 71.1874,Z 101,A 38.9421,B 24.9248,C -2.0032,E1 25.1157,E2 406.53} C_DIS
LIN {X 75.0942,Y 68.7902,Z 101,A 37.4282,B 24.924,C -2.0126,E1 25.1185,E2 408.0149} C_DIS
LIN {X 77.2519,Y 66.3591,Z 101,A 35.4226,B 24.9249,C -2.0014,E1 25.1222,E2 410.038} C_DIS
LIN {X 79.4534,Y 63.7075,Z 101,A 33.2614,B 24.9259,C -1.9879,E1 25.1261,E2 412.2209} C_DIS
LIN {X 82.4007,Y 59.8456,Z 101,A 29.9782,B 24.928,C -1.9594,E1 25.1316,E2 415.5557} C_DIS
LIN {X 85.159,Y 55.85,Z 101,A 28.5373,B 24.9247,C -2.0039,E1 25.1337,E2 416.8844} C_DIS
LIN {X 87.1926,Y 52.6191,Z 101,A 26.042,B 24.9262,C -1.9842,E1 25.1374,E2 419.4135} C_DIS
LIN {X 90.0555,Y 47.5525,Z 101,A 22.7313,B 24.927,C -1.9739,E1 25.1419,E2 422.7315} C_DIS
LIN {X 91.5641,Y 44.5815,Z 101,A 20.1023,B 24.9296,C -1.9383,E1 25.1452,E2 425.4303} C_DIS
LIN {X 93.424,Y 40.5365,Z 101,A 18.3793,B 24.9278,C -1.9626,E1 25.1471,E2 427.0867} C_DIS
LIN {X 94.657,Y 37.5687,Z 101,A 16.4998,B 24.9284,C -1.9544,E1 25.1491,E2 428.9751} C_DIS
LIN {X 95.9248,Y 34.2039,Z 101,A 14.3464,B 24.9292,C -1.9431,E1 25.1511,E2 431.143} C_DIS
LIN {X 97.2127,Y 30.3472,Z 101,A 11.6251,B 24.931,C -1.9188,E1 25.1535,E2 433.9063} C_DIS
LIN {X 98.3689,Y 26.3594,Z 101,A 10.2157,B 24.9288,C -1.9492,E1 25.1545,E2 435.2359} C_DIS
LIN {X 99.5207,Y 21.6067,Z 101,A 7.3617,B 24.9297,C -1.9364,E1 25.1563,E2 438.1034} C_DIS
LIN {X 100.042,Y 19.0491,Z 101,A 5.2188,B 24.932,C -1.9044,E1 25.1575,E2 440.3093} C_DIS
LIN {X 100.6735,Y 15.3654,Z 101,A 3.7647,B 24.9306,C -1.9242,E1 25.1581,E2 441.7083} C_DIS
LIN {X 101.1435,Y 11.8833,Z 101,A 1.8198,B 24.9309,C -1.9192,E1 25.1588,E2 443.6534} C_DIS
LIN {X 101.4716,Y 8.6615,Z 101,A -0.1387,B 24.9318,C -1.9078,E1 25.1593,E2 445.6273} C_DIS
LIN {X 101.71,Y 5.1497,Z 101,A -2.2384,B 24.9326,C -1.8966,E1 25.1597,E2 447.7409} C_DIS
LIN {X 101.8338,Y 1.1876,Z 101,A -4.1522,B 24.9322,C -1.9023,E1 25.1597,E2 449.6298} C_DIS
LIN {X 101.8265,Y -1.6279,Z 101,A -5.8693,B 24.9329,C -1.8918,E1 25.1597,E2 451.3616} C_DIS
LIN {X 101.7186,Y -4.9884,Z 101,A -7.7081,B 24.9332,C -1.8878,E1 25.1595,E2 453.1988} C_DIS
LIN {X 101.4967,Y -8.3487,Z 101,A -9.8315,B 24.9343,C -1.8723,E1 25.1591,E2 455.3461} C_DIS
LIN {X 101.1948,Y -11.4455,Z 101,A -11.4365,B 24.9343,C -1.8726,E1 25.1586,E2 456.9409} C_DIS
LIN {X 100.6945,Y -15.2298,Z 101,A -13.9297,B 24.9357,C -1.8516,E1 25.1576,E2 459.469} C_DIS
LIN {X 100.1264,Y -18.6083,Z 101,A -15.3945,B 24.9349,C -1.8642,E1 25.1569,E2 460.8954} C_DIS
LIN {X 98.9076,Y -24.2596,Z 101,A -18.1496,B 24.9341,C -1.8743,E1 25.1553,E2 463.6107} C_DIS
LIN {X 97.9334,Y -27.9337,Z 101,A -21.121,B 24.937,C -1.8334,E1 25.153,E2 466.6616} C_DIS
LIN {X 96.0009,Y -33.9872,Z 101,A -24.1767,B 24.9363,C -1.8434,E1 25.1504,E2 469.6765} C_DIS
LIN {X 95.0142,Y -36.6593,Z 101,A -26.7529,B 24.9394,C -1.7988,E1 25.1477,E2 472.3434} C_DIS
LIN {X 93.1214,Y -41.2304,Z 101,A -28.5018,B 24.9371,C -1.8323,E1 25.1459,E2 474.0038} C_DIS
LIN {X 91.3598,Y -44.9964,Z 101,A -31.0027,B 24.938,C -1.8187,E1 25.1429,E2 476.5233} C_DIS
LIN {X 89.1829,Y -49.1724,Z 101,A -33.5314,B 24.9382,C -1.8158,E1 25.1396,E2 479.0456} C_DIS
LIN {X 86.5256,Y -53.7087,Z 101,A -36.4508,B 24.9387,C -1.8088,E1 25.1354,E2 481.9665} C_DIS
LIN {X 84.1893,Y -57.3013,Z 101,A -38.8035,B 24.939,C -1.8043,E1 25.1318,E2 484.3179} C_DIS
LIN {X 82.771,Y -59.3316,Z 101,A -40.4242,B 24.9399,C -1.7913,E1 25.1291,E2 485.9616} C_DIS
LIN {X 79.8002,Y -63.2706,Z 101,A -43.3028,B 24.9406,C -1.7796,E1 25.1242,E2 488.854} C_DIS
LIN {X 75.9098,Y -67.889,Z 101,A -47.1357,B 24.9424,C -1.7534,E1 25.1171,E2 492.7316} C_DIS
LIN {X 73.0534,Y -70.9538,Z 101,A -48.6892,B 24.9406,C -1.7798,E1 25.1142,E2 494.2161} C_DIS
LIN {X 70.9639,Y -73.0437,Z 101,A -51.1617,B 24.943,C -1.7433,E1 25.1091,E2 496.7644} C_DIS
LIN {X 67.8302,Y -75.9624,Z 101,A -53.4183,B 24.943,C -1.7438,E1 25.1045,E2 499.0108} C_DIS
LIN {X 64.9952,Y -78.4019,Z 101,A -54.944,B 24.9418,C -1.7621,E1 25.1013,E2 500.4873} C_DIS
LIN {X 61.2309,Y -81.3757,Z 101,A -58.407,B 24.9442,C -1.726,E1 25.0935,E2 504.023} C_DIS
LIN {X 57.4963,Y -84.0573,Z 101,A -60.0607,B 24.9421,C -1.7577,E1 25.0899,E2 505.5962} C_DIS
LIN {X 54.2636,Y -86.179,Z 101,A -62.1666,B 24.9421,C -1.7562,E1 25.085,E2 507.6986} C_DIS
LIN {X 50.415,Y -88.4854,Z 101,A -64.8554,B 24.9429,C -1.745,E1 25.0784,E2 510.4056} C_DIS
LIN {X 47.2291,Y -90.2258,Z 101,A -67.4848,B 24.9447,C -1.7184,E1 25.0718,E2 513.0906} C_DIS
LIN {X 43.908,Y -91.8877,Z 101,A -69.1365,B 24.9438,C -1.7322,E1 25.0678,E2 514.7052} C_DIS
LIN {X 40.5676,Y -93.4104,Z 101,A -71.1277,B 24.9438,C -1.7319,E1 25.0627,E2 516.6921} C_DIS
LIN {X 35.264,Y -95.5396,Z 101,A -74.303,B 24.944,C -1.729,E1 25.0544,E2 519.8672} C_DIS
LIN {X 32.2816,Y -96.5877,Z 101,A -76.8566,B 24.946,C -1.6968,E1 25.0475,E2 522.4923} C_DIS
LIN {X 27.814,Y -97.9674,Z 101,A -78.4706,B 24.9437,C -1.7331,E1 25.0434,E2 524.0174} C_DIS
LIN {X 25.2973,Y -98.6472,Z 101,A -80.1017,B 24.9442,C -1.7252,E1 25.039,E2 525.6648} C_DIS
LIN {X 21.9717,Y -99.4411,Z 101,A -82.7098,B 24.946,C -1.697,E1 25.0317,E2 528.336} C_DIS
LIN {X 17.9774,Y -100.2399,Z 101,A -84.3652,B 24.9446,C -1.7196,E1 25.0273,E2 529.9362} C_DIS
LIN {X 13.263,Y -100.972,Z 101,A -86.8052,B 24.9441,C -1.7271,E1 25.0206,E2 532.3562} C_DIS
LIN {X 10.7049,Y -101.275,Z 101,A -88.4926,B 24.9447,C -1.7171,E1 25.0159,E2 534.0661} C_DIS
LIN {X 7.2471,Y -101.5817,Z 101,A -90.641,B 24.9453,C -1.7086,E1 25.0098,E2 536.2333} C_DIS
LIN {X 2.4666,Y -101.811,Z 101,A -93.215,B 24.9451,C -1.7122,E1 25.0027,E2 538.7983} C_DIS
LIN {X 2.4666,Y -101.811,Z 101,A -93.215,B 24.9451,C -1.7122,E1 25.0027,E2 538.7983} C_DIS
Enddeposition()
LIN {X 0.6996,Y -100.9666,Z 101,A -93.3768,B 24.942,C -1.7588,E1 25.0025,E2 538.8494} C_DIS
Startdeposition()
$VEL.CP = VEL_PRINT
LIN {X 5.3325,Y -100.8287,Z 101,A -90.1338,B 24.9404,C -1.7834,E1 25.0117,E2 535.5491} C_DIS
LIN {X 9.0627,Y -100.5621,Z 101,A -88.5215,B 24.9416,C -1.7647,E1 25.0161,E2 533.982} C_DIS
LIN {X 12.7196,Y -100.1653,Z 101,A -85.7413,B 24.9397,C -1.793,E1 25.024,E2 531.137} C_DIS
LIN {X 17.1874,Y -99.4972,Z 101,A -84.0327,B 24.9418,C -1.7616,E1 25.0285,E2 529.5045} C_DIS
LIN {X 24.1865,Y -98.0301,Z 101,A -79.9903,B 24.9416,C -1.7645,E1 25.0395,E2 525.4604} C_DIS
LIN {X 28.7281,Y -96.7962,Z 101,A -76.6881,B 24.9398,C -1.7923,E1 25.0485,E2 522.0979} C_DIS
LIN {X 32.1767,Y -95.7052,Z 101,A -75.2191,B 24.9412,C -1.7718,E1 25.0523,E2 520.6803} C_DIS
LIN {X 34.9757,Y -94.7189,Z 101,A -73.4065,B 24.9407,C -1.7791,E1 25.0571,E2 518.8543} C_DIS
LIN {X 41.7227,Y -91.9462,Z 101,A -69.3127,B 24.9404,C -1.7833,E1 25.0676,E2 514.7602} C_DIS
LIN {X 44.629,Y -90.5711,Z 101,A -66.8349,B 24.9384,C -1.8123,E1 25.074,E2 512.2202} C_DIS
LIN {X 48.4777,Y -88.5713,Z 101,A -65.0017,B 24.9398,C -1.7914,E1 25.0784,E2 510.4417} C_DIS
LIN {X 51.6996,Y -86.7301,Z 101,A -62.8875,B 24.9396,C -1.7956,E1 25.0835,E2 508.324} C_DIS
LIN {X 57.23,Y -83.1852,Z 101,A -58.9882,B 24.9386,C -1.8098,E1 25.0926,E2 504.4041} C_DIS
LIN {X 62.812,Y -79.054,Z 101,A -55.4452,B 24.9391,C -1.8021,E1 25.1004,E2 500.8921} C_DIS
LIN {X 65.2663,Y -77.0402,Z 101,A -53.2924,B 24.9379,C -1.8204,E1 25.1051,E2 498.7045} C_DIS
LIN {X 69.4478,Y -73.293,Z 101,A -50.1332,B 24.9374,C -1.8268,E1 25.1116,E2 495.543} C_DIS
LIN {X 72.1436,Y -70.6422,Z 101,A -48.2149,B 24.9377,C -1.8228,E1 25.1153,E2 493.6423} C_DIS
LIN {X 75.2765,Y -67.2924,Z 101,A -45.4326,B 24.9368,C -1.8367,E1 25.1206,E2 490.8394} C_DIS
LIN {X 79.0343,Y -62.8369,Z 101,A -42.6406,B 24.9376,C -1.8244,E1 25.1255,E2 488.0893} C_DIS
LIN {X 81.9528,Y -58.9807,Z 101,A -39.6368,B 24.9364,C -1.8424,E1 25.1306,E2 485.0574} C_DIS
LIN {X 85.2916,Y -54.0418,Z 101,A -36.384,B 24.9361,C -1.8465,E1 25.1356,E2 481.811} C_DIS
LIN {X 87.443,Y -50.4835,Z 101,A -33.8281,B 24.9351,C -1.8614,E1 25.1393,E2 479.2331} C_DIS
LIN {X 91.0628,Y -43.6165,Z 101,A -30.0427,B 24.9359,C -1.849,E1 25.1441,E2 475.4969} C_DIS
LIN {X 92.7139,Y -39.9888,Z 101,A -26.7678,B 24.9325,C -1.8975,E1 25.1479,E2 472.1254} C_DIS
LIN {X 94.1268,Y -36.5393,Z 101,A -25.148,B 24.9335,C -1.8835,E1 25.1496,E2 470.5476} C_DIS
LIN {X 95.2384,Y -33.5332,Z 101,A -23.5435,B 24.9337,C -1.8804,E1 25.1511,E2 468.9595} C_DIS
LIN {X 97.1457,Y -27.5231,Z 101,A -19.707,B 24.9322,C -1.9022,E1 25.1542,E2 465.0933} C_DIS
LIN {X 98.2421,Y -23.3143,Z 101,A -16.7094,B 24.93,C -1.932,E1 25.1562,E2 462.0427} C_DIS
LIN {X 99.1308,Y -19.1808,Z 101,A -15.3866,B 24.9327,C -1.8952,E1 25.1569,E2 460.8144} C_DIS
LIN {X 100.0141,Y -13.8603,Z 101,A -11.9011,B 24.9307,C -1.9225,E1 25.1585,E2 457.2851} C_DIS
LIN {X 100.6456,Y -8.0795,Z 101,A -8.421,B 24.9294,C -1.9406,E1 25.1594,E2 453.783} C_DIS
LIN {X 100.9104,Y -3.4701,Z 101,A -6.0642,B 24.9296,C -1.9382,E1 25.1597,E2 451.4458} C_DIS
LIN {X 100.9708,Y 0.0838,Z 101,A -3.7501,B 24.9282,C -1.957,E1 25.1597,E2 449.1012} C_DIS
LIN {X 100.8277,Y 5.3515,Z 101,A -1.1187,B 24.9286,C -1.9518,E1 25.1595,E2 446.4977} C_DIS
LIN {X 100.6081,Y 8.5488,Z 101,A 0.6884,B 24.9282,C -1.9571,E1 25.1591,E2 444.6887} C_DIS
LIN {X 100.3641,Y 11.0527,Z 101,A 2.5609,B 24.9265,C -1.98,E1 25.1585,E2 442.7734} C_DIS
LIN {X 99.9448,Y 14.3479,Z 101,A 3.6746,B 24.9284,C -1.9542,E1 25.1581,E2 441.727} C_DIS
LIN {X 98.8534,Y 20.5643,Z 101,A 7.248,B 24.9276,C -1.965,E1 25.1564,E2 438.1489} C_DIS
LIN {X 97.6047,Y 25.853,Z 101,A 11.1025,B 24.9245,C -2.0061,E1 25.1537,E2 434.2199} C_DIS
LIN {X 96.6162,Y 29.3338,Z 101,A 12.6962,B 24.9255,C -1.9934,E1 25.1525,E2 432.6652} C_DIS
LIN {X 95.5517,Y 32.6318,Z 101,A 14.7452,B 24.9248,C -2.0027,E1 25.1507,E2 430.6059} C_DIS
LIN {X 94.1569,Y 36.4626,Z 101,A 16.987,B 24.9245,C -2.0066,E1 25.1484,E2 428.3674} C_DIS
LIN {X 92.4521,Y 40.5892,Z 101,A 20.2862,B 24.9216,C -2.0453,E1 25.1447,E2 424.9949} C_DIS
LIN {X 90.3111,Y 45.1536,Z 101,A 22.1392,B 24.9241,C -2.0121,E1 25.1425,E2 423.2302} C_DIS
LIN {X 89.0326,Y 47.624,Z 101,A 24.3337,B 24.9219,C -2.0415,E1 25.1396,E2 420.9779} C_DIS
LIN {X 87.2263,Y 50.86,Z 101,A 25.951,B 24.9229,C -2.0274,E1 25.1374,E2 419.4022} C_DIS
LIN {X 85.5771,Y 53.5852,Z 101,A 27.6764,B 24.9229,C -2.0288,E1 25.1349,E2 417.6821} C_DIS
LIN {X 84.3265,Y 55.5325,Z 101,A 29.53,B 24.9209,C -2.0541,E1 25.1319,E2 415.7782} C_DIS
LIN {X 82.276,Y 58.5277,Z 101,A 31.178,B 24.9218,C -2.0426,E1 25.1293,E2 414.1653} C_DIS
LIN {X 80.0575,Y 61.5274,Z 101,A 33.1321,B 24.9218,C -2.0412,E1 25.1261,E2 412.2237} C_DIS
LIN {X 77.9633,Y 64.1621,Z 101,A 35.0809,B 24.9214,C -2.0473,E1 25.1226,E2 410.2697} C_DIS
LIN {X 75.9211,Y 66.5645,Z 101,A 36.812,B 24.9213,C -2.0491,E1 25.1195,E2 408.542} C_DIS
LIN {X 73.3367,Y 69.402,Z 101,A 39.0947,B 24.9206,C -2.0582,E1 25.1151,E2 406.2481} C_DIS
LIN {X 70.745,Y 72.042,Z 101,A 41.1358,B 24.9204,C -2.0603,E1 25.1111,E2 404.2105} C_DIS
LIN {X 68.3518,Y 74.3159,Z 101,A 42.95,B 24.9203,C -2.0618,E1 25.1074,E2 402.4002} C_DIS
LIN {X 65.8285,Y 76.5613,Z 101,A 44.8174,B 24.9201,C -2.0636,E1 25.1035,E2 400.5358} C_DIS
LIN {X 63.2858,Y 78.6746,Z 101,A 47.3245,B 24.9179,C -2.0922,E1 25.0979,E2 397.9708} C_DIS
LIN {X 60.1575,Y 81.0941,Z 101,A 49.0214,B 24.9193,C -2.0745,E1 25.0942,E2 396.3219} C_DIS
LIN {X 57.2881,Y 83.1448,Z 101,A 51.1975,B 24.9185,C -2.0847,E1 25.0892,E2 394.129} C_DIS
LIN {X 53.8315,Y 85.4233,Z 101,A 53.4823,B 24.9185,C -2.0859,E1 25.0839,E2 391.8489} C_DIS
LIN {X 50.5768,Y 87.3893,Z 101,A 56.201,B 24.9164,C -2.111,E1 25.0772,E2 389.0789} C_DIS
LIN {X 46.6943,Y 89.5236,Z 101,A 58.2218,B 24.9177,C -2.095,E1 25.0723,E2 387.1017} C_DIS
LIN {X 43.562,Y 91.089,Z 101,A 60.3041,B 24.9172,C -2.1012,E1 25.067,E2 385.0103} C_DIS
LIN {X 38.8317,Y 93.2045,Z 101,A 62.9884,B 24.9177,C -2.0944,E1 25.0602,E2 382.3484} C_DIS
LIN {X 35.5374,Y 94.5091,Z 101,A 64.7838,B 24.9182,C -2.0881,E1 25.0556,E2 380.5718} C_DIS
LIN {X 31.2104,Y 96.0247,Z 101,A 67.664,B 24.9172,C -2.101,E1 25.0479,E2 377.6667} C_DIS
LIN {X 27.3759,Y 97.1874,Z 101,A 69.6664,B 24.9179,C -2.0923,E1 25.0426,E2 375.6885} C_DIS
LIN {X 24.5251,Y 97.9472,Z 101,A 71.3495,B 24.9178,C -2.0936,E1 25.0381,E2 374.0048} C_DIS
LIN {X 18.6244,Y 99.2379,Z 101,A 74.685,B 24.9179,C -2.0917,E1 25.029,E2 370.678} C_DIS
LIN {X 13.7208,Y 100.0339,Z 101,A 77.5727,B 24.9177,C -2.0951,E1 25.021,E2 367.7851} C_DIS
LIN {X 9.4291,Y 100.5282,Z 101,A 80.0932,B 24.9174,C -2.0981,E1 25.014,E2 365.2593} C_DIS
LIN {X 6.3084,Y 100.7734,Z 101,A 81.7739,B 24.9177,C -2.0946,E1 25.0093,E2 363.5877} C_DIS
LIN {X 2.6905,Y 100.9342,Z 101,A 84.1735,B 24.9167,C -2.1073,E1 25.0025,E2 361.1586} C_DIS
LIN {X -1.6595,Y 100.9559,Z 101,A 86.3909,B 24.9175,C -2.0974,E1 24.9964,E2 358.9646} C_DIS
LIN {X -4.8796,Y 100.8529,Z 101,A 88.8461,B 24.9157,C -2.1201,E1 24.9894,E2 356.455} C_DIS
LIN {X -8.7314,Y 100.5924,Z 101,A 90.739,B 24.9167,C -2.108,E1 24.9842,E2 354.5899} C_DIS
LIN {X -14.47,Y 99.9275,Z 101,A 93.4501,B 24.9185,C -2.0852,E1 24.9769,E2 351.9311} C_DIS
LIN {X -21.4057,Y 98.6743,Z 101,A 97.3795,B 24.9189,C -2.0795,E1 24.9661,E2 348.0112} C_DIS
LIN {X -26.4233,Y 97.4507,Z 101,A 100.6811,B 24.9181,C -2.09,E1 24.9571,E2 344.6799} C_DIS
LIN {X -29.9116,Y 96.4371,Z 101,A 102.8609,B 24.9179,C -2.092,E1 24.9512,E2 342.4917} C_DIS
LIN {X -33.868,Y 95.1209,Z 101,A 105.1669,B 24.9183,C -2.0869,E1 24.9451,E2 340.1934} C_DIS
LIN {X -36.8747,Y 93.9951,Z 101,A 106.6953,B 24.9193,C -2.0739,E1 24.9412,E2 338.6926} C_DIS
LIN {X -38.9732,Y 93.1448,Z 101,A 108.4547,B 24.9181,C -2.0891,E1 24.9366,E2 336.893} C_DIS
LIN {X -43.2748,Y 91.227,Z 101,A 110.9203,B 24.9191,C -2.0776,E1 24.9304,E2 334.4487} C_DIS
LIN {X -46.0182,Y 89.873,Z 101,A 112.6099,B 24.9194,C -2.0732,E1 24.9262,E2 332.7652} C_DIS
LIN {X -50.0518,Y 87.691,Z 101,A 115.6235,B 24.9186,C -2.0833,E1 24.9187,E2 329.7188} C_DIS
LIN {X -54.137,Y 85.2305,Z 101,A 117.816,B 24.9204,C -2.0601,E1 24.9137,E2 327.5748} C_DIS
LIN {X -56.7922,Y 83.4834,Z 101,A 120.2531,B 24.9189,C -2.079,E1 24.9079,E2 325.0846} C_DIS
LIN {X -59.532,Y 81.5523,Z 101,A 121.8412,B 24.9201,C -2.0639,E1 24.9044,E2 323.5267} C_DIS
LIN {X -62.9243,Y 78.9652,Z 101,A 124.1046,B 24.9209,C -2.0532,E1 24.8994,E2 321.2805} C_DIS
LIN {X -67.4783,Y 75.11,Z 101,A 127.4312,B 24.9217,C -2.0435,E1 24.8924,E2 317.9641} C_DIS
LIN {X -69.11,Y 73.6114,Z 101,A 129.2325,B 24.9205,C -2.0596,E1 24.8886,E2 316.117} C_DIS
LIN {X -71.4834,Y 71.3105,Z 101,A 130.7462,B 24.9218,C -2.0424,E1 24.8857,E2 314.638} C_DIS
LIN {X -75.3167,Y 67.2475,Z 101,A 133.7939,B 24.9227,C -2.0302,E1 24.8799,E2 311.6059} C_DIS
LIN {X -77.2187,Y 65.0565,Z 101,A 135.7494,B 24.9222,C -2.0367,E1 24.8764,E2 309.6261} C_DIS
LIN {X -79.8889,Y 61.7462,Z 101,A 138.2458,B 24.9225,C -2.0332,E1 24.872,E2 307.1263} C_DIS
LIN {X -83.1455,Y 57.2871,Z 101,A 142.0693,B 24.9213,C -2.0487,E1 24.8658,E2 303.2471} C_DIS
LIN {X -86.0175,Y 52.8779,Z 101,A 144.1663,B 24.9243,C -2.0093,E1 24.8629,E2 301.2333} C_DIS
LIN {X -88.6168,Y 48.3938,Z 101,A 147.4914,B 24.9239,C -2.014,E1 24.8583,E2 297.8796} C_DIS
LIN {X -90.1107,Y 45.5529,Z 101,A 148.9852,B 24.9252,C -1.9973,E1 24.8564,E2 296.4177} C_DIS
Enddeposition()
END
